# B&R Automation Studio project PT_KB_V01 (part 4)

#### FBAI01_DI01_DO2.st
```iecst
FUNCTION_BLOCK FBAI01_DI01_DO02 (* Skaliranje transmitera sa AI + status DI + 2 DO izbora opsega *) (*$GROUP=User,$CAT=User,$GROUPICON=User.png,$CATICON=User.png*)

(* -------------------------------------------------------------------------- *)
(* 1) Podrazumevane vrednosti po scan-u                                        *)
(* -------------------------------------------------------------------------- *)
(* Podrazumevane vrednosti po scan-u. *)
AI_Output.Status := FALSE;
AI_Internal.FaultCondition := FALSE;
AI_Internal.FaultProcess := FALSE;
AI_Internal.FaultConfig := FALSE;
AI_Output.UnitOfMeasureOut := AI_Param.UnitOfMeasure;
AI_Output.TransmitterStatusIn := AI_Input.TransmitterStatus;
AI_Output.RangeChanging := FALSE;
AI_Output.FaultProcessOut := FALSE;
AI_Output.FaultConfigOut := FALSE;
AI_Internal.ResetRequest := AI_Input.ResetAlarm;

(* -------------------------------------------------------------------------- *)
(* 2) Reset i detekcija promene opsega                                         *)
(* -------------------------------------------------------------------------- *)
(* Eksplicitni reset latched alarma. *)
IF AI_Internal.ResetRequest THEN
	AI_Internal.FaultLatched := FALSE;
END_IF;

(* Detekcija promene opsega. *)
IF AI_Input.RangeSelect <> AI_Internal.PrevRangeSelect THEN
	AI_Internal.RangeChangeMem := TRUE;
END_IF;

(* -------------------------------------------------------------------------- *)
(* 3) Izbor opsega i mapiranje DO bitova                                       *)
(* -------------------------------------------------------------------------- *)
(* Izbor aktivnog opsega i mapiranje u 2 izlazna DO bita. *)
CASE AI_Input.RangeSelect OF
	1:
		AI_Output.ActiveRange := 1;
		AI_Output.RangeBit0_out := FALSE;
		AI_Output.RangeBit1_out := FALSE;
		AI_Internal.ActiveScaledMin := AI_Param.ScaledMin_R1;
		AI_Internal.ActiveScaledMax := AI_Param.ScaledMax_R1;
		AI_Output.RangeComment := 'Opseg 1';
	2:
		AI_Output.ActiveRange := 2;
		AI_Output.RangeBit0_out := TRUE;
		AI_Output.RangeBit1_out := FALSE;
		AI_Internal.ActiveScaledMin := AI_Param.ScaledMin_R2;
		AI_Internal.ActiveScaledMax := AI_Param.ScaledMax_R2;
		AI_Output.RangeComment := 'Opseg 2';
	3:
		AI_Output.ActiveRange := 3;
		AI_Output.RangeBit0_out := FALSE;
		AI_Output.RangeBit1_out := TRUE;
		AI_Internal.ActiveScaledMin := AI_Param.ScaledMin_R3;
		AI_Internal.ActiveScaledMax := AI_Param.ScaledMax_R3;
		AI_Output.RangeComment := 'Opseg 3';
	4:
		AI_Output.ActiveRange := 4;
		AI_Output.RangeBit0_out := TRUE;
		AI_Output.RangeBit1_out := TRUE;
		AI_Internal.ActiveScaledMin := AI_Param.ScaledMin_R4;
		AI_Internal.ActiveScaledMax := AI_Param.ScaledMax_R4;
		AI_Output.RangeComment := 'Opseg 4';
	ELSE
		AI_Output.ActiveRange := 1;
		AI_Output.RangeBit0_out := FALSE;
		AI_Output.RangeBit1_out := FALSE;
		AI_Internal.ActiveScaledMin := AI_Param.ScaledMin_R1;
		AI_Internal.ActiveScaledMax := AI_Param.ScaledMax_R1;
		AI_Output.RangeComment := 'Nevalidan opseg';
		AI_Internal.FaultConfig := TRUE;
END_CASE;

(* -------------------------------------------------------------------------- *)
(* 4) Ogranicenje manual vrednosti i range-settle tajmer                       *)
(* -------------------------------------------------------------------------- *)
(* Ogranicenje manual vrednosti na aktivni opseg. *)
AI_Internal.ManualValueLimited := AI_Input.ManualValue;
IF AI_Internal.ManualValueLimited < AI_Internal.ActiveScaledMin THEN
	AI_Internal.ManualValueLimited := AI_Internal.ActiveScaledMin;
END_IF;
IF AI_Internal.ManualValueLimited > AI_Internal.ActiveScaledMax THEN
	AI_Internal.ManualValueLimited := AI_Internal.ActiveScaledMax;
END_IF;

(* Tajmer stabilizacije nakon promene opsega. *)
AI_Internal.RangeSettleTimeEffective := AI_Input.RangeSettleTime;
IF AI_Internal.RangeSettleTimeEffective <= T#0ms THEN
	AI_Internal.RangeSettleTimeEffective := T#2s;
	AI_Internal.FaultConfig := TRUE;
END_IF;

AI_Internal.RangeSettleTimer(
	IN := AI_Internal.RangeChangeMem,
	PT := AI_Internal.RangeSettleTimeEffective
);
AI_Output.RangeChanging := AI_Internal.RangeChangeMem;
IF AI_Internal.RangeSettleTimer.Q THEN
	AI_Internal.RangeChangeMem := FALSE;
END_IF;

(* -------------------------------------------------------------------------- *)
(* 5) Glavna obrada kada je blok omogucen                                      *)
(* -------------------------------------------------------------------------- *)
IF NOT AI_Input.Enable THEN
	AI_Output.ScaledValue := 0.0;
	AI_Output.State := AI_Constant.ST_DISABLED;
	AI_Output.State_comment := AI_Constant.CMT_DISABLED;
	AI_Output.Status := FALSE;
ELSE
	(* Racunanje raspona za linearnu transformaciju raw -> scaled. *)
	AI_Internal.ScaleSpanRaw := INT_TO_REAL(AI_Param.RawMax - AI_Param.RawMin);
	AI_Internal.ScaleSpanScaled := AI_Internal.ActiveScaledMax - AI_Internal.ActiveScaledMin;

	IF AI_Internal.ScaleSpanRaw <= 0.0 THEN
		AI_Internal.FaultConfig := TRUE;
	END_IF;

	IF AI_Internal.ScaleSpanScaled <= 0.0 THEN
		AI_Internal.FaultConfig := TRUE;
	END_IF;

	IF AI_Input.ManualAlarm THEN
		AI_Internal.FaultProcess := TRUE;
	END_IF;

	IF NOT AI_Output.RangeChanging THEN
		IF AI_Input.UnderRange OR AI_Input.OverRange THEN
			AI_Internal.FaultProcess := TRUE;
		END_IF;

		IF NOT AI_Input.TransmitterStatus THEN
			AI_Internal.FaultProcess := TRUE;
		END_IF;
	END_IF;

	IF AI_Output.RangeChanging THEN
		AI_Output.ScaledValue := AI_Internal.LastGoodScaledValue;
	ELSIF AI_Input.EnableManual THEN
		AI_Output.ScaledValue := AI_Internal.ManualValueLimited;
		AI_Internal.LastGoodScaledValue := AI_Output.ScaledValue;
	ELSE
		IF AI_Internal.ScaleSpanRaw > 0.0 THEN
			AI_Output.ScaledValue :=
				AI_Internal.ActiveScaledMin +
				((INT_TO_REAL(AI_Input.RawValue - AI_Param.RawMin) / AI_Internal.ScaleSpanRaw) * AI_Internal.ScaleSpanScaled);
			AI_Internal.LastGoodScaledValue := AI_Output.ScaledValue;
		ELSE
			AI_Output.ScaledValue := AI_Internal.ActiveScaledMin;
		END_IF;
	END_IF;

	AI_Internal.FaultCondition := AI_Internal.FaultProcess OR AI_Internal.FaultConfig;
	AI_Output.FaultProcessOut := AI_Internal.FaultProcess;
	AI_Output.FaultConfigOut := AI_Internal.FaultConfig;

	IF AI_Internal.FaultCondition THEN
		AI_Internal.FaultLatched := TRUE;
	END_IF;

	(* ---------------------------------------------------------------------- *)
	(* 6) State i status mapiranje                                             *)
	(* ---------------------------------------------------------------------- *)
	IF AI_Output.RangeChanging THEN
		AI_Output.State := AI_Constant.ST_RANGE_CHANGING;
		AI_Output.State_comment := AI_Constant.CMT_RANGE_CHANGING;
		AI_Output.Status := FALSE;
	ELSIF AI_Internal.FaultLatched AND AI_Input.EnableManual THEN
		AI_Output.State := AI_Constant.ST_MANUAL_FAULT;
		AI_Output.State_comment := AI_Constant.CMT_MANUAL_FAULT;
		AI_Output.Status := FALSE;
	ELSIF AI_Input.EnableManual THEN
		AI_Output.State := AI_Constant.ST_MANUAL;
		AI_Output.State_comment := AI_Constant.CMT_MANUAL;
		AI_Output.Status := AI_Input.TransmitterStatus;
	ELSIF AI_Internal.FaultLatched THEN
		AI_Output.State := AI_Constant.ST_FAULT;
		AI_Output.State_comment := AI_Constant.CMT_FAULT;
		AI_Output.Status := FALSE;
	ELSIF NOT AI_Input.TransmitterStatus THEN
		AI_Output.State := AI_Constant.ST_TRANSMITTER_STATUS_0;
		AI_Output.State_comment := AI_Constant.CMT_TRANSMITTER_STATUS_0;
		AI_Output.Status := FALSE;
	ELSIF AI_Input.RawValue < AI_Param.RawMin THEN
		AI_Output.State := AI_Constant.ST_UNDERRANGE;
		AI_Output.State_comment := AI_Constant.CMT_UNDERRANGE;
		AI_Output.Status := FALSE;
	ELSIF AI_Input.RawValue > AI_Param.RawMax THEN
		AI_Output.State := AI_Constant.ST_OVERRANGE;
		AI_Output.State_comment := AI_Constant.CMT_OVERRANGE;
		AI_Output.Status := FALSE;
	ELSE
		AI_Output.State := AI_Constant.ST_ACTIVE;
		AI_Output.State_comment := AI_Constant.CMT_ACTIVE;
		AI_Output.Status := TRUE;
	END_IF;
END_IF;

(* -------------------------------------------------------------------------- *)
(* 7) Pamcenje prethodnog opsega za sledeci scan                               *)
(* -------------------------------------------------------------------------- *)
(* Pamcenje prethodnog opsega. *)
AI_Internal.PrevRangeSelect := AI_Input.RangeSelect;

END_FUNCTION_BLOCK
```

#### FB_PvAiAo_Fast.st
```iecst
FUNCTION_BLOCK FB_PvAiAo_Fast

(* Preporuka za commissioning (nije automatsko prepisivanje parametara):
	DeviationOnLimit = 8.0
	DeviationOffLimit = 3.0
	DeviationTime = T#5s
*)

(* -------------------------------------------------------------------------- *)
(* 1) Osnovni statusi bloka                                                    *)
(* -------------------------------------------------------------------------- *)
PV_Output.Valid := PV_Input.Enable;
PV_Output.ManualActive := PV_Input.EnableManual;

(* -------------------------------------------------------------------------- *)
(* 2) Ogranicenje AI ulaza i skaliranje u procente                             *)
(* -------------------------------------------------------------------------- *)
IF PV_Input.AI_Raw < PV_Constant.RAW_MIN THEN
	PV_Output.AI_Raw_Limited := PV_Constant.RAW_MIN;
ELSIF PV_Input.AI_Raw > PV_Constant.RAW_MAX THEN
	PV_Output.AI_Raw_Limited := PV_Constant.RAW_MAX;
ELSE
	PV_Output.AI_Raw_Limited := PV_Input.AI_Raw;
END_IF;

PV_Internal.rAi := INT_TO_REAL(PV_Output.AI_Raw_Limited);
PV_Output.PV_Percent := (PV_Internal.rAi * PV_Constant.PCT_MAX) / INT_TO_REAL(PV_Constant.RAW_MAX);

(* -------------------------------------------------------------------------- *)
(* 3) Ogranicenje auto i manual komande                                        *)
(* -------------------------------------------------------------------------- *)
IF PV_Input.SP_Percent < PV_Constant.PCT_MIN THEN
	PV_Output.SP_Percent_Limited := PV_Constant.PCT_MIN;
ELSIF PV_Input.SP_Percent > PV_Constant.PCT_MAX THEN
	PV_Output.SP_Percent_Limited := PV_Constant.PCT_MAX;
ELSE
	PV_Output.SP_Percent_Limited := PV_Input.SP_Percent;
END_IF;

IF PV_Input.ManualValue_Percent < PV_Constant.PCT_MIN THEN
	PV_Output.ManualValue_Limited := PV_Constant.PCT_MIN;
ELSIF PV_Input.ManualValue_Percent > PV_Constant.PCT_MAX THEN
	PV_Output.ManualValue_Limited := PV_Constant.PCT_MAX;
ELSE
	PV_Output.ManualValue_Limited := PV_Input.ManualValue_Percent;
END_IF;

(* -------------------------------------------------------------------------- *)
(* 4) Izbor aktivne komande (manual ima prioritet)                             *)
(* -------------------------------------------------------------------------- *)
IF PV_Input.EnableManual THEN
	PV_Output.ActiveSP_Limited := PV_Output.ManualValue_Limited;
ELSE
	PV_Output.ActiveSP_Limited := PV_Output.SP_Percent_Limited;
END_IF;
PV_Output.ActiveSP_Percent := PV_Output.ActiveSP_Limited;

(* -------------------------------------------------------------------------- *)
(* 5) Validacija devijacionih granica i vremena                                *)
(* -------------------------------------------------------------------------- *)
IF PV_Param.DeviationOnLimit < PV_Constant.PCT_MIN THEN
	PV_Output.DeviationOn_Limited := PV_Constant.PCT_MIN;
ELSIF PV_Param.DeviationOnLimit > PV_Constant.PCT_MAX THEN
	PV_Output.DeviationOn_Limited := PV_Constant.PCT_MAX;
ELSE
	PV_Output.DeviationOn_Limited := PV_Param.DeviationOnLimit;
END_IF;

IF PV_Param.DeviationOffLimit < PV_Constant.PCT_MIN THEN
	PV_Output.DeviationOff_Limited := PV_Constant.PCT_MIN;
ELSIF PV_Param.DeviationOffLimit > PV_Constant.PCT_MAX THEN
	PV_Output.DeviationOff_Limited := PV_Constant.PCT_MAX;
ELSE
	PV_Output.DeviationOff_Limited := PV_Param.DeviationOffLimit;
END_IF;

IF PV_Output.DeviationOff_Limited > PV_Output.DeviationOn_Limited THEN
	PV_Output.DeviationOff_Limited := PV_Output.DeviationOn_Limited;
END_IF;

IF PV_Param.DeviationTime <= T#0ms THEN
	PV_Output.DeviationTime_Effective := PV_Constant.MIN_DEV_TIME;
ELSE
	PV_Output.DeviationTime_Effective := PV_Param.DeviationTime;
END_IF;

(* -------------------------------------------------------------------------- *)
(* 6) Proracun devijacije i tolerancije                                        *)
(* -------------------------------------------------------------------------- *)
PV_Output.DeviationPercent := ABS(PV_Output.ActiveSP_Limited - PV_Output.PV_Percent);
PV_Output.InTolerance := (PV_Output.DeviationPercent <= PV_Output.DeviationOff_Limited);

(* -------------------------------------------------------------------------- *)
(* 7) Fault/reset/deviation stanje i tajmer                                     *)
(* -------------------------------------------------------------------------- *)
IF PV_Input.Reset THEN
	PV_Output.FaultActive := FALSE;
	PV_Output.DeviationTimeout := FALSE;
	PV_Output.InDeviation := FALSE;

	PV_Internal.FB_DeviationTimer.PT := PV_Output.DeviationTime_Effective;
	PV_Internal.FB_DeviationTimer.IN := FALSE;
	PV_Internal.FB_DeviationTimer();
	PV_Output.DeviationElapsed := PV_Internal.FB_DeviationTimer.ET;

ELSIF NOT PV_Input.Enable THEN
	PV_Output.InDeviation := FALSE;

	PV_Internal.FB_DeviationTimer.PT := PV_Output.DeviationTime_Effective;
	PV_Internal.FB_DeviationTimer.IN := FALSE;
	PV_Internal.FB_DeviationTimer();
	PV_Output.DeviationElapsed := PV_Internal.FB_DeviationTimer.ET;

ELSE
	IF PV_Output.FaultActive THEN
		PV_Output.InDeviation := FALSE;

		PV_Internal.FB_DeviationTimer.PT := PV_Output.DeviationTime_Effective;
		PV_Internal.FB_DeviationTimer.IN := FALSE;
		PV_Internal.FB_DeviationTimer();
		PV_Output.DeviationElapsed := PV_Internal.FB_DeviationTimer.ET;
	ELSE
		IF NOT PV_Output.InDeviation THEN
			IF PV_Output.DeviationPercent >= PV_Output.DeviationOn_Limited THEN
				PV_Output.InDeviation := TRUE;
			END_IF;
		ELSE
			IF PV_Output.DeviationPercent <= PV_Output.DeviationOff_Limited THEN
				PV_Output.InDeviation := FALSE;
			END_IF;
		END_IF;

		PV_Internal.FB_DeviationTimer.PT := PV_Output.DeviationTime_Effective;
		PV_Internal.FB_DeviationTimer.IN := PV_Output.InDeviation;
		PV_Internal.FB_DeviationTimer();
		PV_Output.DeviationElapsed := PV_Internal.FB_DeviationTimer.ET;

		IF PV_Output.InDeviation AND PV_Internal.FB_DeviationTimer.Q THEN
			PV_Output.FaultActive := TRUE;
			PV_Output.DeviationTimeout := TRUE;
			PV_Output.InDeviation := FALSE;
		END_IF;
	END_IF;
END_IF;

(* -------------------------------------------------------------------------- *)
(* 8) Izbor stvarno primenjene izlazne komande                                  *)
(* -------------------------------------------------------------------------- *)
IF NOT PV_Input.Enable THEN
	PV_Output.AppliedOutput_Limited := PV_Constant.PCT_MIN;
	PV_Output.FrozenOutput_Percent := PV_Constant.PCT_MIN;
	PV_Output.CommandPermitted := FALSE;
	PV_Output.ForceActive := FALSE;

ELSIF PV_Output.FaultActive THEN
	IF PV_Input.ForceCmd THEN
		PV_Output.AppliedOutput_Limited := PV_Output.ActiveSP_Limited;
		PV_Output.CommandPermitted := TRUE;
		PV_Output.ForceActive := TRUE;
	ELSE
		PV_Output.CommandPermitted := FALSE;
		PV_Output.ForceActive := FALSE;

		IF PV_Param.HoldOutputOnFault THEN
			PV_Output.AppliedOutput_Limited := PV_Output.FrozenOutput_Percent;
		ELSE
			PV_Output.AppliedOutput_Limited := PV_Constant.PCT_MIN;
		END_IF;
	END_IF;
ELSE
	PV_Output.AppliedOutput_Limited := PV_Output.ActiveSP_Limited;
	PV_Output.CommandPermitted := TRUE;
	PV_Output.ForceActive := FALSE;
	PV_Output.FrozenOutput_Percent := PV_Output.AppliedOutput_Limited;
END_IF;

(* -------------------------------------------------------------------------- *)
(* 9) Zavrsno ogranicenje i AO skaliranje                                      *)
(* -------------------------------------------------------------------------- *)
IF PV_Output.AppliedOutput_Limited < PV_Constant.PCT_MIN THEN
	PV_Output.AppliedOutput_Limited := PV_Constant.PCT_MIN;
ELSIF PV_Output.AppliedOutput_Limited > PV_Constant.PCT_MAX THEN
	PV_Output.AppliedOutput_Limited := PV_Constant.PCT_MAX;
END_IF;
PV_Output.AppliedOutput_Percent := PV_Output.AppliedOutput_Limited;

PV_Internal.rAo := (PV_Output.AppliedOutput_Limited * INT_TO_REAL(PV_Constant.RAW_MAX)) / PV_Constant.PCT_MAX;
PV_Internal.AO_Raw_Calc := REAL_TO_INT(PV_Internal.rAo);

IF PV_Internal.AO_Raw_Calc < PV_Constant.RAW_MIN THEN
	PV_Internal.AO_Raw_Calc := PV_Constant.RAW_MIN;
ELSIF PV_Internal.AO_Raw_Calc > PV_Constant.RAW_MAX THEN
	PV_Internal.AO_Raw_Calc := PV_Constant.RAW_MAX;
END_IF;
PV_Output.AO_Raw := PV_Internal.AO_Raw_Calc;

(* -------------------------------------------------------------------------- *)
(* 10) Standardni izlazi stanja za HMI/SCADA                                    *)
(* -------------------------------------------------------------------------- *)
IF NOT PV_Input.Enable THEN
	PV_Output.Status := FALSE;
	PV_Output.State := PV_Constant.ST_DISABLED;
	PV_Output.State_comment := 'ST_DISABLED - blok nije omogucen';
ELSIF PV_Output.FaultActive THEN
	PV_Output.Status := FALSE;
	IF PV_Output.ForceActive THEN
		PV_Output.State := PV_Constant.ST_FAULT_FORCE;
		PV_Output.State_comment := 'ST_FAULT_FORCE - fault aktivan, izlaz forsiran';
	ELSE
		PV_Output.State := PV_Constant.ST_FAULT_HOLD;
		PV_Output.State_comment := 'ST_FAULT_HOLD - fault aktivan, izlaz blokiran/hold';
	END_IF;
ELSIF PV_Output.InDeviation THEN
	PV_Output.Status := TRUE;
	PV_Output.State := PV_Constant.ST_DEVIATION_ACTIVE;
	PV_Output.State_comment := 'ST_DEVIATION_ACTIVE - aktivno pracenje devijacije';
ELSIF PV_Output.ManualActive THEN
	PV_Output.Status := TRUE;
	PV_Output.State := PV_Constant.ST_MANUAL_ACTIVE;
	PV_Output.State_comment := 'ST_MANUAL_ACTIVE - aktivan manuelni rezim';
ELSE
	PV_Output.Status := TRUE;
	PV_Output.State := PV_Constant.ST_AUTO_ACTIVE;
	PV_Output.State_comment := 'ST_AUTO_ACTIVE - aktivan automatski rezim';
END_IF;

END_FUNCTION_BLOCK
```

#### FB_PvAiAo_Slow.st
```iecst
(* SLOW VARIJANTA: Za elektromotorne ventile sa sporim odzivom (30-180 s). *)
(* Implementirana logika: trenutna komanda + nadzor fizickog pracenja ventila. *)

(*
===============================================================================
SLOW LOGIC SPEC (USAGLASENO PRE IMPLEMENTACIJE)
===============================================================================

Osnovni princip:
1) Komanda izlaza se NE rampira softverski.
2) Kada se promeni setpoint, izlaz odmah dobija novu komandnu vrednost.
3) Umesto rampe proverava se da li ventil fizicki prati ocekivano vreme putovanja.

Definicije:
- PV_Internal.StepDeltaPercent = ABS(NewSP - PV_Internal.PrevSP)
- Smer kretanja:
	- Opening: NewSP > PV_Internal.PrevSP
	- Closing: NewSP < PV_Internal.PrevSP
- Ocekivano vreme putovanja:
	- Texp_open  = PV_Internal.StepDeltaPercent/100 * PV_Internal.TravelTimeOpenFull
	- Texp_close = PV_Internal.StepDeltaPercent/100 * PV_Internal.TravelTimeCloseFull
- Dozvoljeni prozor:
	- Tmin = Texp * (1 - PV_Internal.TimeTolerancePercent/100)
	- Tmax = Texp * (1 + PV_Internal.TimeTolerancePercent/100)

Ulaz u tracking poteza:
- Tracking se aktivira kada je ABS(NewSP - PV_Internal.PrevSP) >= StepMinPercent.
- Ako je manji korak od StepMinPercent, tretira se kao mali pomak bez punog timing nadzora.

Uslovi tokom tracking-a:
1) Start movement timeout:
	 - Ako nema detektovanog pocetnog pomeranja PV u PV_Internal.StartMoveTimeout -> FaultNoMovement.
2) Smer kretanja:
	 - Opening: PV mora da raste.
	 - Closing: PV mora da opada.
	 - Suprotan smer duze od PV_Internal.DirectionCheckTime -> FaultWrongDirection.
3) Stall nadzor:
	 - Ako je tracking aktivan, a PV ne menja vrednost duze od PV_Internal.StallTimeout -> FaultStall.
4) Zavrsetak poteza:
	 - Potez je zavrsen kada PV udje u ciljnu traku:
		 ABS(TargetSP - PV) <= TargetBandPercent.
	 - Ako zavrsetak nastupi pre Tmin -> warning ili fault (po parametru PV_Internal.EnableTooFastFault).
	 - Ako zavrsetak ne nastupi do Tmax -> FaultTimeout.

Nova komanda tokom aktivnog poteza:
- Aktivni tracking se prekida i odmah se formira novi tracking od trenutnog PV/SP stanja.

Fault politika:
- Fault je latched (ostaje aktivan do Reset).
- Fault tipovi:
	1) NoMovement
	2) WrongDirection
	3) Stall
	4) TimeoutSlow
	5) (opciono) TooFast

Interakcija sa postojecim logikama:
- Enable i dalje ima apsolutni prioritet (disable gasi komandu).
- ForceCmd i HoldOutputOnFault zadrzavaju isto ponasanje kao FAST varijanta.
- Status/State/State_comment ostaju obavezni izlazi.

Napomena za implementaciju:
- Uvesti odvojene interne tajmere za:
	- start movement timeout,
	- direction confirm,
	- stall timeout,
	- tracking timeout (Tmax).
- Uvesti internu memoriju prethodnog SP i prethodnog PV za detekciju koraka i trenda.
===============================================================================
*)

FUNCTION_BLOCK FB_PvAiAo_Slow

(* Commissioning preset (pocetne preporuke, po potrebi menjati na terenu):
   PV_Internal.TravelTimeOpenFull = T#120s
   PV_Internal.TravelTimeCloseFull = T#120s
   PV_Internal.TimeTolerancePercent = 35.0
   PV_Internal.StartMoveTimeout = T#8s
   PV_Internal.DirectionCheckTime = T#8s
   PV_Internal.StallTimeout = T#20s
   PV_Internal.MovementStartDeltaPercent = 0.7
   PV_Internal.PerScanProgressMinPercent = 0.03
   PV_Internal.DirectionEpsPercent = 0.03
   PV_Internal.EnableTooFastFault = FALSE
*)

(* -------------------------------------------------------------------------- *)
(* 1) Osnovni statusi bloka                                                    *)
(* -------------------------------------------------------------------------- *)
PV_Output.Valid := PV_Input.Enable;
PV_Output.ManualActive := PV_Input.EnableManual;

(* -------------------------------------------------------------------------- *)
(* 2) Ogranicenje AI ulaza i skaliranje u procente                             *)
(* -------------------------------------------------------------------------- *)
IF PV_Input.AI_Raw < PV_Constant.RAW_MIN THEN
	PV_Output.AI_Raw_Limited := PV_Constant.RAW_MIN;
ELSIF PV_Input.AI_Raw > PV_Constant.RAW_MAX THEN
	PV_Output.AI_Raw_Limited := PV_Constant.RAW_MAX;
ELSE
	PV_Output.AI_Raw_Limited := PV_Input.AI_Raw;
END_IF;

PV_Internal.rAi := INT_TO_REAL(PV_Output.AI_Raw_Limited);
PV_Output.PV_Percent := (PV_Internal.rAi * PV_Constant.PCT_MAX) / INT_TO_REAL(PV_Constant.RAW_MAX);

(* -------------------------------------------------------------------------- *)
(* 3) Ogranicenje auto i manual komande                                        *)
(* -------------------------------------------------------------------------- *)
IF PV_Input.SP_Percent < PV_Constant.PCT_MIN THEN
	PV_Output.SP_Percent_Limited := PV_Constant.PCT_MIN;
ELSIF PV_Input.SP_Percent > PV_Constant.PCT_MAX THEN
	PV_Output.SP_Percent_Limited := PV_Constant.PCT_MAX;
ELSE
	PV_Output.SP_Percent_Limited := PV_Input.SP_Percent;
END_IF;

IF PV_Input.ManualValue_Percent < PV_Constant.PCT_MIN THEN
	PV_Output.ManualValue_Limited := PV_Constant.PCT_MIN;
ELSIF PV_Input.ManualValue_Percent > PV_Constant.PCT_MAX THEN
	PV_Output.ManualValue_Limited := PV_Constant.PCT_MAX;
ELSE
	PV_Output.ManualValue_Limited := PV_Input.ManualValue_Percent;
END_IF;

(* -------------------------------------------------------------------------- *)
(* 4) Izbor aktivne komande (manual ima prioritet)                             *)
(* -------------------------------------------------------------------------- *)
IF PV_Input.EnableManual THEN
	PV_Output.ActiveSP_Limited := PV_Output.ManualValue_Limited;
ELSE
	PV_Output.ActiveSP_Limited := PV_Output.SP_Percent_Limited;
END_IF;
PV_Output.ActiveSP_Percent := PV_Output.ActiveSP_Limited;

(* -------------------------------------------------------------------------- *)
(* 5) Validacija devijacionih granica i vremena                                *)
(* -------------------------------------------------------------------------- *)
IF PV_Param.DeviationOnLimit < PV_Constant.PCT_MIN THEN
	PV_Output.DeviationOn_Limited := PV_Constant.PCT_MIN;
ELSIF PV_Param.DeviationOnLimit > PV_Constant.PCT_MAX THEN
	PV_Output.DeviationOn_Limited := PV_Constant.PCT_MAX;
ELSE
	PV_Output.DeviationOn_Limited := PV_Param.DeviationOnLimit;
END_IF;

IF PV_Param.DeviationOffLimit < PV_Constant.PCT_MIN THEN
	PV_Output.DeviationOff_Limited := PV_Constant.PCT_MIN;
ELSIF PV_Param.DeviationOffLimit > PV_Constant.PCT_MAX THEN
	PV_Output.DeviationOff_Limited := PV_Constant.PCT_MAX;
ELSE
	PV_Output.DeviationOff_Limited := PV_Param.DeviationOffLimit;
END_IF;

IF PV_Output.DeviationOff_Limited > PV_Output.DeviationOn_Limited THEN
	PV_Output.DeviationOff_Limited := PV_Output.DeviationOn_Limited;
END_IF;

IF PV_Param.DeviationTime <= T#0ms THEN
	PV_Output.DeviationTime_Effective := PV_Constant.MIN_DEV_TIME;
ELSE
	PV_Output.DeviationTime_Effective := PV_Param.DeviationTime;
END_IF;

(* -------------------------------------------------------------------------- *)
(* 6) Proracun devijacije i tolerancije                                        *)
(* -------------------------------------------------------------------------- *)
PV_Output.DeviationPercent := ABS(PV_Output.ActiveSP_Limited - PV_Output.PV_Percent);
PV_Output.InTolerance := (PV_Output.DeviationPercent <= PV_Output.DeviationOff_Limited);

(* -------------------------------------------------------------------------- *)
(* 7) Tracking i fault nadzor za SLOW ponasanje                                *)
(* -------------------------------------------------------------------------- *)
(* Reset/safe defaults za tracking i fault nadzor. *)
IF PV_Input.Reset THEN
	PV_Output.FaultActive := FALSE;
	PV_Output.DeviationTimeout := FALSE;
	PV_Internal.TrackActive := FALSE;
	PV_Internal.MovementStarted := FALSE;
	PV_Internal.FaultReasonText := 'RESET';
	PV_Output.InDeviation := FALSE;

	PV_Internal.TrackTimer(IN := FALSE, PT := T#1ms);
	PV_Internal.StartMoveTimer(IN := FALSE, PT := PV_Internal.StartMoveTimeout);
	PV_Internal.DirectionTimer(IN := FALSE, PT := PV_Internal.DirectionCheckTime);
	PV_Internal.StallTimer(IN := FALSE, PT := PV_Internal.StallTimeout);

ELSIF NOT PV_Input.Enable THEN
	PV_Internal.TrackActive := FALSE;
	PV_Internal.MovementStarted := FALSE;
	PV_Output.InDeviation := FALSE;
	PV_Internal.FaultReasonText := 'DISABLED';

	PV_Internal.TrackTimer(IN := FALSE, PT := T#1ms);
	PV_Internal.StartMoveTimer(IN := FALSE, PT := PV_Internal.StartMoveTimeout);
	PV_Internal.DirectionTimer(IN := FALSE, PT := PV_Internal.DirectionCheckTime);
	PV_Internal.StallTimer(IN := FALSE, PT := PV_Internal.StallTimeout);

ELSE
	(* Novo pracenje na znacajnu promenu komande.
	   Prag za aktivaciju tracking-a je vezan za DeviationOn_Limited. *)
	PV_Internal.StepDeltaPercent := ABS(PV_Output.ActiveSP_Limited - PV_Internal.PrevSP);
	IF PV_Internal.StepDeltaPercent >= PV_Output.DeviationOn_Limited THEN
		PV_Internal.TrackActive := TRUE;
		PV_Internal.MovementStarted := FALSE;
		PV_Internal.PV_AtTrackStart := PV_Output.PV_Percent;
		PV_Internal.LastProgressPV := PV_Output.PV_Percent;
		PV_Internal.TrackDirectionOpen := (PV_Output.ActiveSP_Limited > PV_Internal.PrevSP);

		IF PV_Internal.TrackDirectionOpen THEN
			PV_Internal.ExpectedTravelSec := (PV_Internal.StepDeltaPercent / 100.0) * (TIME_TO_REAL(PV_Internal.TravelTimeOpenFull) / 1000.0);
		ELSE
			PV_Internal.ExpectedTravelSec := (PV_Internal.StepDeltaPercent / 100.0) * (TIME_TO_REAL(PV_Internal.TravelTimeCloseFull) / 1000.0);
		END_IF;

		PV_Internal.TminSec := PV_Internal.ExpectedTravelSec * (1.0 - PV_Internal.TimeTolerancePercent / 100.0);
		PV_Internal.TmaxSec := PV_Internal.ExpectedTravelSec * (1.0 + PV_Internal.TimeTolerancePercent / 100.0);
		IF PV_Internal.TminSec < 0.0 THEN
			PV_Internal.TminSec := 0.0;
		END_IF;
		IF PV_Internal.TmaxSec <= 0.0 THEN
			PV_Internal.TmaxSec := 0.1;
		END_IF;
	END_IF;

	(* Tajmeri nadzora putovanja. *)
	PV_Internal.TrackTimer(IN := PV_Internal.TrackActive, PT := REAL_TO_TIME(PV_Internal.TmaxSec * 1000.0));
	PV_Internal.StartMoveTimer(IN := PV_Internal.TrackActive AND (NOT PV_Internal.MovementStarted), PT := PV_Internal.StartMoveTimeout);

	IF PV_Internal.TrackActive THEN
		IF ABS(PV_Output.PV_Percent - PV_Internal.PV_AtTrackStart) >= PV_Internal.MovementStartDeltaPercent THEN
			PV_Internal.MovementStarted := TRUE;
		END_IF;

		IF PV_Internal.TrackDirectionOpen THEN
			PV_Internal.DirectionTimer(IN := (PV_Output.PV_Percent < (PV_Internal.PrevPV - PV_Internal.DirectionEpsPercent)), PT := PV_Internal.DirectionCheckTime);
		ELSE
			PV_Internal.DirectionTimer(IN := (PV_Output.PV_Percent > (PV_Internal.PrevPV + PV_Internal.DirectionEpsPercent)), PT := PV_Internal.DirectionCheckTime);
		END_IF;

		PV_Internal.StallTimer(IN := PV_Internal.MovementStarted AND (ABS(PV_Output.PV_Percent - PV_Internal.PrevPV) < PV_Internal.PerScanProgressMinPercent), PT := PV_Internal.StallTimeout);
	ELSE
		PV_Internal.DirectionTimer(IN := FALSE, PT := PV_Internal.DirectionCheckTime);
		PV_Internal.StallTimer(IN := FALSE, PT := PV_Internal.StallTimeout);
	END_IF;

	(* Fault uslovi i zavrsetak tracking-a. *)
	PV_Output.DeviationTimeout := FALSE;
	IF PV_Internal.TrackActive THEN
		IF PV_Internal.StartMoveTimer.Q THEN
			PV_Output.FaultActive := TRUE;
			PV_Internal.FaultReasonText := 'FAULT_NO_MOVEMENT';
			PV_Internal.TrackActive := FALSE;
		ELSIF PV_Internal.DirectionTimer.Q THEN
			PV_Output.FaultActive := TRUE;
			PV_Internal.FaultReasonText := 'FAULT_WRONG_DIRECTION';
			PV_Internal.TrackActive := FALSE;
		ELSIF PV_Internal.StallTimer.Q THEN
			PV_Output.FaultActive := TRUE;
			PV_Internal.FaultReasonText := 'FAULT_STALL';
			PV_Internal.TrackActive := FALSE;
		ELSIF PV_Internal.TrackTimer.Q THEN
			PV_Output.FaultActive := TRUE;
			PV_Output.DeviationTimeout := TRUE;
			PV_Internal.FaultReasonText := 'FAULT_TIMEOUT_SLOW';
			PV_Internal.TrackActive := FALSE;
		ELSIF PV_Output.InTolerance THEN
			PV_Internal.ActualTravelSec := TIME_TO_REAL(PV_Internal.TrackTimer.ET) / 1000.0;
			IF PV_Internal.EnableTooFastFault AND (PV_Internal.ActualTravelSec < PV_Internal.TminSec) THEN
				PV_Output.FaultActive := TRUE;
				PV_Internal.FaultReasonText := 'FAULT_TOO_FAST';
			ELSE
				PV_Internal.FaultReasonText := 'TRACK_OK';
			END_IF;
			PV_Internal.TrackActive := FALSE;
		END_IF;
	END_IF;

	PV_Output.InDeviation := PV_Internal.TrackActive;
END_IF;

PV_Output.DeviationElapsed := PV_Internal.TrackTimer.ET;

(* -------------------------------------------------------------------------- *)
(* 8) Izbor stvarno primenjene izlazne komande                                  *)
(* -------------------------------------------------------------------------- *)
(* Immediate command (bez rampe), sa istom fault politikom kao FAST. *)
IF NOT PV_Input.Enable THEN
	PV_Output.AppliedOutput_Limited := PV_Constant.PCT_MIN;
	PV_Output.FrozenOutput_Percent := PV_Constant.PCT_MIN;
	PV_Output.CommandPermitted := FALSE;
	PV_Output.ForceActive := FALSE;

ELSIF PV_Output.FaultActive THEN
	IF PV_Input.ForceCmd THEN
		PV_Output.AppliedOutput_Limited := PV_Output.ActiveSP_Limited;
		PV_Output.CommandPermitted := TRUE;
		PV_Output.ForceActive := TRUE;
	ELSE
		PV_Output.CommandPermitted := FALSE;
		PV_Output.ForceActive := FALSE;
		IF PV_Param.HoldOutputOnFault THEN
			PV_Output.AppliedOutput_Limited := PV_Output.FrozenOutput_Percent;
		ELSE
			PV_Output.AppliedOutput_Limited := PV_Constant.PCT_MIN;
		END_IF;
	END_IF;

ELSE
	PV_Output.AppliedOutput_Limited := PV_Output.ActiveSP_Limited;
	PV_Output.CommandPermitted := TRUE;
	PV_Output.ForceActive := FALSE;
	PV_Output.FrozenOutput_Percent := PV_Output.AppliedOutput_Limited;
END_IF;

(* -------------------------------------------------------------------------- *)
(* 9) Zavrsno ogranicenje i AO skaliranje                                      *)
(* -------------------------------------------------------------------------- *)
IF PV_Output.AppliedOutput_Limited < PV_Constant.PCT_MIN THEN
	PV_Output.AppliedOutput_Limited := PV_Constant.PCT_MIN;
ELSIF PV_Output.AppliedOutput_Limited > PV_Constant.PCT_MAX THEN
	PV_Output.AppliedOutput_Limited := PV_Constant.PCT_MAX;
END_IF;

PV_Output.AppliedOutput_Percent := PV_Output.AppliedOutput_Limited;
PV_Internal.rAo := (PV_Output.AppliedOutput_Limited * INT_TO_REAL(PV_Constant.RAW_MAX)) / PV_Constant.PCT_MAX;
PV_Internal.AO_Raw_Calc := REAL_TO_INT(PV_Internal.rAo);
IF PV_Internal.AO_Raw_Calc < PV_Constant.RAW_MIN THEN
	PV_Internal.AO_Raw_Calc := PV_Constant.RAW_MIN;
ELSIF PV_Internal.AO_Raw_Calc > PV_Constant.RAW_MAX THEN
	PV_Internal.AO_Raw_Calc := PV_Constant.RAW_MAX;
END_IF;
PV_Output.AO_Raw := PV_Internal.AO_Raw_Calc;

(* -------------------------------------------------------------------------- *)
(* 10) Standardni izlazi stanja za HMI/SCADA                                    *)
(* -------------------------------------------------------------------------- *)
IF NOT PV_Input.Enable THEN
	PV_Output.Status := FALSE;
	PV_Output.State := PV_Constant.ST_DISABLED;
	PV_Output.State_comment := 'ST_DISABLED - blok nije omogucen';
ELSIF PV_Output.FaultActive THEN
	PV_Output.Status := FALSE;
	IF PV_Output.ForceActive THEN
		PV_Output.State := PV_Constant.ST_FAULT_FORCE;
		PV_Output.State_comment := CONCAT('ST_FAULT_FORCE - ', PV_Internal.FaultReasonText);
	ELSE
		PV_Output.State := PV_Constant.ST_FAULT_HOLD;
		PV_Output.State_comment := CONCAT('ST_FAULT_HOLD - ', PV_Internal.FaultReasonText);
	END_IF;
ELSIF PV_Output.InDeviation THEN
	PV_Output.Status := TRUE;
	PV_Output.State := PV_Constant.ST_DEVIATION_ACTIVE;
	PV_Output.State_comment := 'ST_DEVIATION_ACTIVE - tracking travel time';
ELSIF PV_Output.ManualActive THEN
	PV_Output.Status := TRUE;
	PV_Output.State := PV_Constant.ST_MANUAL_ACTIVE;
	PV_Output.State_comment := 'ST_MANUAL_ACTIVE - aktivan manuelni rezim';
ELSE
	PV_Output.Status := TRUE;
	PV_Output.State := PV_Constant.ST_AUTO_ACTIVE;
	PV_Output.State_comment := 'ST_AUTO_ACTIVE - aktivan automatski rezim';
END_IF;

(* -------------------------------------------------------------------------- *)
(* 11) Memorija prethodnog ciklusa za detekciju koraka i trenda                 *)
(* -------------------------------------------------------------------------- *)
PV_Internal.PrevSP := PV_Output.ActiveSP_Limited;
PV_Internal.PrevPV := PV_Output.PV_Percent;

END_FUNCTION_BLOCK
```

#### FB_PvAoNoFb.st
```iecst
FUNCTION_BLOCK FB_PvAoNoFb

(* -------------------------------------------------------------------------- *)
(* 1) Osnovni statusi i izbor rezima                                           *)
(* -------------------------------------------------------------------------- *)
PV_Output.ManualActive := PV_Input.ManualMode;
PV_Output.ForceActive := FALSE;
PV_Output.ParamInvalid := FALSE;

(* -------------------------------------------------------------------------- *)
(* 2) Validacija parametara i priprema efektivnih granica                      *)
(* -------------------------------------------------------------------------- *)
IF (PV_Param.OutMin < PV_Constant.PCT_MIN) OR
   (PV_Param.OutMin > PV_Constant.PCT_MAX) OR
   (PV_Param.OutMax < PV_Constant.PCT_MIN) OR
   (PV_Param.OutMax > PV_Constant.PCT_MAX) OR
   (PV_Param.OutMin >= PV_Param.OutMax) OR
   (PV_Param.RampUp < 0.0) OR
   (PV_Param.RampDown < 0.0) OR
   (PV_Param.OnDelay < T#0ms) OR
   (PV_Param.OffDelay < T#0ms) THEN
	PV_Output.ParamInvalid := TRUE;
END_IF;

IF PV_Output.ParamInvalid THEN
	PV_Output.OutMin_Effective := PV_Constant.PCT_MIN;
	PV_Output.OutMax_Effective := PV_Constant.PCT_MAX;
	PV_Output.RampUp_Effective := PV_Constant.PCT_MAX;
	PV_Output.RampDown_Effective := PV_Constant.PCT_MAX;
	PV_Output.OnDelay_Effective := T#0ms;
	PV_Output.OffDelay_Effective := T#0ms;
ELSE
	PV_Output.OutMin_Effective := PV_Param.OutMin;
	PV_Output.OutMax_Effective := PV_Param.OutMax;

	IF PV_Param.RampUp <= PV_Constant.STEP_MIN THEN
		PV_Output.RampUp_Effective := PV_Constant.PCT_MAX;
	ELSE
		PV_Output.RampUp_Effective := PV_Param.RampUp;
	END_IF;

	IF PV_Param.RampDown <= PV_Constant.STEP_MIN THEN
		PV_Output.RampDown_Effective := PV_Constant.PCT_MAX;
	ELSE
		PV_Output.RampDown_Effective := PV_Param.RampDown;
	END_IF;

	PV_Output.OnDelay_Effective := PV_Param.OnDelay;
	PV_Output.OffDelay_Effective := PV_Param.OffDelay;
END_IF;

(* -------------------------------------------------------------------------- *)
(* 3) Fault latch i reset politika                                              *)
(* -------------------------------------------------------------------------- *)
IF PV_Input.ResetFault AND NOT PV_Output.ParamInvalid THEN
	PV_Output.FaultActive := FALSE;
	PV_Output.FaultCode := PV_Constant.FLT_NONE;
END_IF;

IF PV_Output.ParamInvalid THEN
	PV_Output.FaultActive := TRUE;
	PV_Output.FaultCode := PV_Constant.FLT_PARAM_INVALID;
END_IF;

IF NOT PV_Input.Enable THEN
	PV_Output.ForceActive := FALSE;
END_IF;

(* -------------------------------------------------------------------------- *)
(* 4) Izbor i ogranicenje komandnog cilja                                       *)
(* -------------------------------------------------------------------------- *)
IF PV_Input.ManualMode THEN
	PV_Output.CmdTarget := PV_Input.ManualOut;
ELSE
	PV_Output.CmdTarget := PV_Input.AutoSP;
END_IF;

IF PV_Output.CmdTarget < PV_Constant.PCT_MIN THEN
	PV_Output.CmdTarget := PV_Constant.PCT_MIN;
ELSIF PV_Output.CmdTarget > PV_Constant.PCT_MAX THEN
	PV_Output.CmdTarget := PV_Constant.PCT_MAX;
END_IF;

PV_Output.CmdLimited := PV_Output.CmdTarget;
IF PV_Output.CmdLimited < PV_Output.OutMin_Effective THEN
	PV_Output.CmdLimited := PV_Output.OutMin_Effective;
ELSIF PV_Output.CmdLimited > PV_Output.OutMax_Effective THEN
	PV_Output.CmdLimited := PV_Output.OutMax_Effective;
END_IF;

(* -------------------------------------------------------------------------- *)
(* 5) OnDelay/OffDelay logika bez feedback-a                                   *)
(* -------------------------------------------------------------------------- *)
PV_Internal.RiseRequest := (PV_Output.CmdLimited > (PV_Output.OutMin_Effective + PV_Internal.EpsPercent));
PV_Internal.FallRequest := NOT PV_Internal.RiseRequest;

PV_Internal.OnDelayTimer(IN := (PV_Input.Enable AND PV_Internal.RiseRequest), PT := PV_Output.OnDelay_Effective);
PV_Internal.OffDelayTimer(IN := (PV_Input.Enable AND PV_Internal.FallRequest), PT := PV_Output.OffDelay_Effective);

IF NOT PV_Input.Enable THEN
	PV_Output.CmdDelayed := PV_Constant.PCT_MIN;
ELSIF PV_Internal.RiseRequest THEN
	IF (PV_Output.OnDelay_Effective <= T#0ms) OR PV_Internal.OnDelayTimer.Q THEN
		PV_Output.CmdDelayed := PV_Output.CmdLimited;
	ELSE
		PV_Output.CmdDelayed := PV_Output.OutMin_Effective;
	END_IF;
ELSE
	IF (PV_Output.OffDelay_Effective <= T#0ms) OR PV_Internal.OffDelayTimer.Q THEN
		PV_Output.CmdDelayed := PV_Output.OutMin_Effective;
	ELSE
		PV_Output.CmdDelayed := PV_Internal.CmdWorking;
	END_IF;
END_IF;

(* -------------------------------------------------------------------------- *)
(* 6) Fault reakcija i force/hold ponasanje                                    *)
(* -------------------------------------------------------------------------- *)
IF NOT PV_Input.Enable THEN
	PV_Output.CmdDelayed := PV_Constant.PCT_MIN;
	PV_Output.ForceActive := FALSE;
ELSIF PV_Output.FaultActive THEN
	IF PV_Input.ForceCmd THEN
		PV_Output.ForceActive := TRUE;
	ELSE
		PV_Output.ForceActive := FALSE;
		IF PV_Param.HoldOnFault THEN
			PV_Output.CmdDelayed := PV_Internal.LastHealthyCmd;
		ELSE
			PV_Output.CmdDelayed := PV_Output.OutMin_Effective;
		END_IF;
	END_IF;
END_IF;

(* -------------------------------------------------------------------------- *)
(* 7) Ramp limit komande (po ciklusu)                                          *)
(* -------------------------------------------------------------------------- *)
IF NOT PV_Input.Enable THEN
	PV_Internal.CmdWorking := PV_Constant.PCT_MIN;
ELSE
	IF PV_Output.CmdDelayed > PV_Internal.CmdWorking THEN
		PV_Internal.CmdWorking := PV_Internal.CmdWorking + PV_Output.RampUp_Effective;
		IF PV_Internal.CmdWorking > PV_Output.CmdDelayed THEN
			PV_Internal.CmdWorking := PV_Output.CmdDelayed;
		END_IF;
	ELSIF PV_Output.CmdDelayed < PV_Internal.CmdWorking THEN
		PV_Internal.CmdWorking := PV_Internal.CmdWorking - PV_Output.RampDown_Effective;
		IF PV_Internal.CmdWorking < PV_Output.CmdDelayed THEN
			PV_Internal.CmdWorking := PV_Output.CmdDelayed;
		END_IF;
	END_IF;
END_IF;

IF PV_Internal.CmdWorking < PV_Constant.PCT_MIN THEN
	PV_Internal.CmdWorking := PV_Constant.PCT_MIN;
ELSIF PV_Internal.CmdWorking > PV_Constant.PCT_MAX THEN
	PV_Internal.CmdWorking := PV_Constant.PCT_MAX;
END_IF;

PV_Output.AO_Cmd := PV_Internal.CmdWorking;

IF PV_Input.Enable AND NOT PV_Output.FaultActive THEN
	PV_Internal.LastHealthyCmd := PV_Output.AO_Cmd;
END_IF;

(* -------------------------------------------------------------------------- *)
(* 8) Standardni izlazi stanja                                                 *)
(* -------------------------------------------------------------------------- *)
IF NOT PV_Input.Enable THEN
	PV_Output.Status := FALSE;
	PV_Output.State := PV_Constant.ST_DISABLED;
	PV_Output.State_comment := 'ST_DISABLED - blok nije omogucen';
ELSIF PV_Output.FaultActive THEN
	PV_Output.Status := FALSE;
	IF PV_Output.ForceActive THEN
		PV_Output.State := PV_Constant.ST_FAULT_FORCE;
		PV_Output.State_comment := 'ST_FAULT_FORCE - fault aktivan, izlaz forsiran';
	ELSE
		PV_Output.State := PV_Constant.ST_FAULT_HOLD;
		PV_Output.State_comment := 'ST_FAULT_HOLD - fault aktivan, izlaz hold/zero';
	END_IF;
ELSIF PV_Output.ManualActive THEN
	PV_Output.Status := TRUE;
	PV_Output.State := PV_Constant.ST_MANUAL_ACTIVE;
	PV_Output.State_comment := 'ST_MANUAL_ACTIVE - manuelni rezim';
ELSE
	PV_Output.Status := TRUE;
	PV_Output.State := PV_Constant.ST_AUTO_ACTIVE;
	PV_Output.State_comment := 'ST_AUTO_ACTIVE - automatski rezim';
END_IF;

END_FUNCTION_BLOCK
```

#### FB_AirRelease.st
```iecst
FUNCTION_BLOCK FB_AirRelease (* Automatsko odzracivanje cevovoda sa 1 do 3 LS senzora. *)

(* -------------------------------------------------------------------------- *)
(* 1) Runtime vreme task ciklusa                                               *)
(* -------------------------------------------------------------------------- *)
AR_Internal.RtInfo(enable := TRUE);
AR_Internal.RuntimeTimeValid :=
	(AR_Internal.RtInfo.status = 0)
	AND (AR_Internal.RtInfo.cycle_time > 0)
	AND (AR_Internal.RtInfo.cycle_time <= 1000000);

IF AR_Internal.RuntimeTimeValid THEN
	AR_Output.CycleTime_s := UDINT_TO_REAL(AR_Internal.RtInfo.cycle_time) / 1000000.0;
ELSE
	AR_Output.CycleTime_s := 0.0;
END_IF;

(* -------------------------------------------------------------------------- *)
(* 2) Validacija parametara                                                    *)
(* -------------------------------------------------------------------------- *)
AR_Internal.ConfigValid := TRUE;
AR_Internal.ConfigFaultText := 'CONFIG_OK';

IF (AR_Param.NumberOfLS < 1) OR (AR_Param.NumberOfLS > 3) THEN
	AR_Internal.ConfigValid := FALSE;
	AR_Internal.ConfigFaultText := 'NumberOfLS mora biti u opsegu 1..3';
ELSIF AR_Param.PressureSP_bar < 0.0 THEN
	AR_Internal.ConfigValid := FALSE;
	AR_Internal.ConfigFaultText := 'PressureSP_bar ne sme biti negativan';
ELSIF (AR_Param.PressureHysteresis_bar < 0.0)
	OR (AR_Param.PressureHysteresis_bar > AR_Param.PressureSP_bar) THEN
	AR_Internal.ConfigValid := FALSE;
	AR_Internal.ConfigFaultText := 'PressureHysteresis_bar mora biti 0..PressureSP';
ELSIF (AR_Param.LS1.SP_Percent < AR_Constant.PCT_MIN)
	OR (AR_Param.LS1.SP_Percent > AR_Constant.PCT_MAX) THEN
	AR_Internal.ConfigValid := FALSE;
	AR_Internal.ConfigFaultText := 'LS1 SP mora biti u opsegu 0..100%';
ELSIF AR_Param.LS1.Ramp_PercentPerSecond < AR_Constant.RAMP_MIN THEN
	AR_Internal.ConfigValid := FALSE;
	AR_Internal.ConfigFaultText := 'LS1 rampa mora biti veca od 0%/s';
ELSIF (AR_Param.LS1.ConfirmTime_s < 0.0)
	OR (AR_Param.LS1.ConfirmTime_s > AR_Constant.CONFIRM_TIME_MAX_S) THEN
	AR_Internal.ConfigValid := FALSE;
	AR_Internal.ConfigFaultText := 'LS1 ConfirmTime_s mora biti 0..3600 s';
ELSIF (AR_Param.NumberOfLS >= 2)
	AND ((AR_Param.LS2.SP_Percent < AR_Constant.PCT_MIN)
		OR (AR_Param.LS2.SP_Percent > AR_Constant.PCT_MAX)) THEN
	AR_Internal.ConfigValid := FALSE;
	AR_Internal.ConfigFaultText := 'LS2 SP mora biti u opsegu 0..100%';
ELSIF (AR_Param.NumberOfLS >= 2)
	AND (AR_Param.LS2.Ramp_PercentPerSecond < AR_Constant.RAMP_MIN) THEN
	AR_Internal.ConfigValid := FALSE;
	AR_Internal.ConfigFaultText := 'LS2 rampa mora biti veca od 0%/s';
ELSIF (AR_Param.NumberOfLS >= 2)
	AND ((AR_Param.LS2.ConfirmTime_s < 0.0)
		OR (AR_Param.LS2.ConfirmTime_s > AR_Constant.CONFIRM_TIME_MAX_S)) THEN
	AR_Internal.ConfigValid := FALSE;
	AR_Internal.ConfigFaultText := 'LS2 ConfirmTime_s mora biti 0..3600 s';
ELSIF (AR_Param.NumberOfLS >= 2)
	AND (AR_Param.LS2.SP_Percent < AR_Param.LS1.SP_Percent) THEN
	AR_Internal.ConfigValid := FALSE;
	AR_Internal.ConfigFaultText := 'LS2 SP mora biti veci ili jednak LS1 SP';
ELSIF (AR_Param.NumberOfLS = 3)
	AND ((AR_Param.LS3.SP_Percent < AR_Constant.PCT_MIN)
		OR (AR_Param.LS3.SP_Percent > AR_Constant.PCT_MAX)) THEN
	AR_Internal.ConfigValid := FALSE;
	AR_Internal.ConfigFaultText := 'LS3 SP mora biti u opsegu 0..100%';
ELSIF (AR_Param.NumberOfLS = 3)
	AND (AR_Param.LS3.Ramp_PercentPerSecond < AR_Constant.RAMP_MIN) THEN
	AR_Internal.ConfigValid := FALSE;
	AR_Internal.ConfigFaultText := 'LS3 rampa mora biti veca od 0%/s';
ELSIF (AR_Param.NumberOfLS = 3)
	AND ((AR_Param.LS3.ConfirmTime_s < 0.0)
		OR (AR_Param.LS3.ConfirmTime_s > AR_Constant.CONFIRM_TIME_MAX_S)) THEN
	AR_Internal.ConfigValid := FALSE;
	AR_Internal.ConfigFaultText := 'LS3 ConfirmTime_s mora biti 0..3600 s';
ELSIF (AR_Param.NumberOfLS = 3)
	AND (AR_Param.LS3.SP_Percent < AR_Param.LS2.SP_Percent) THEN
	AR_Internal.ConfigValid := FALSE;
	AR_Internal.ConfigFaultText := 'LS3 SP mora biti veci ili jednak LS2 SP';
END_IF;

IF AR_Internal.ConfigValid THEN
	AR_Internal.LS1ConfirmTime := REAL_TO_TIME(AR_Param.LS1.ConfirmTime_s * 1000.0);
	AR_Internal.LS2ConfirmTime := REAL_TO_TIME(AR_Param.LS2.ConfirmTime_s * 1000.0);
	AR_Internal.LS3ConfirmTime := REAL_TO_TIME(AR_Param.LS3.ConfirmTime_s * 1000.0);
ELSE
	AR_Internal.LS1ConfirmTime := T#1s;
	AR_Internal.LS2ConfirmTime := T#1s;
	AR_Internal.LS3ConfirmTime := T#1s;
END_IF;

(* -------------------------------------------------------------------------- *)
(* 3) Dvosmerna vremenska potvrda LS signala                                  *)
(* -------------------------------------------------------------------------- *)
AR_Internal.TonLS1Change.IN :=
	AR_Internal.ConfigValid
	AND (AR_Input.LS1_Upper <> AR_Internal.LS1Confirmed);
AR_Internal.TonLS1Change.PT := AR_Internal.LS1ConfirmTime;
AR_Internal.TonLS1Change();

IF AR_Internal.TonLS1Change.Q THEN
	AR_Internal.LS1Confirmed := AR_Input.LS1_Upper;
END_IF;

IF AR_Param.NumberOfLS >= 2 THEN
	AR_Internal.TonLS2Change.IN :=
		AR_Internal.ConfigValid
		AND (AR_Input.LS2_Middle <> AR_Internal.LS2Confirmed);
	AR_Internal.TonLS2Change.PT := AR_Internal.LS2ConfirmTime;
	AR_Internal.TonLS2Change();

	IF AR_Internal.TonLS2Change.Q THEN
		AR_Internal.LS2Confirmed := AR_Input.LS2_Middle;
	END_IF;
ELSE
	AR_Internal.TonLS2Change(IN := FALSE, PT := T#0ms);
	AR_Internal.LS2Confirmed := FALSE;
END_IF;

IF AR_Param.NumberOfLS = 3 THEN
	AR_Internal.TonLS3Change.IN :=
		AR_Internal.ConfigValid
		AND (AR_Input.LS3_Lower <> AR_Internal.LS3Confirmed);
	AR_Internal.TonLS3Change.PT := AR_Internal.LS3ConfirmTime;
	AR_Internal.TonLS3Change();

	IF AR_Internal.TonLS3Change.Q THEN
		AR_Internal.LS3Confirmed := AR_Input.LS3_Lower;
	END_IF;
ELSE
	AR_Internal.TonLS3Change(IN := FALSE, PT := T#0ms);
	AR_Internal.LS3Confirmed := FALSE;
END_IF;

(* -------------------------------------------------------------------------- *)
(* 4) Monitoring aktivnog pritiska sa histerezom                              *)
(* -------------------------------------------------------------------------- *)
IF NOT AR_Input.Enable OR NOT AR_Internal.ConfigValid THEN
	AR_Internal.PressureActive := FALSE;
ELSIF NOT AR_Internal.PressureActive THEN
	IF AR_Input.Pressure_bar > AR_Param.PressureSP_bar THEN
		AR_Internal.PressureActive := TRUE;
	END_IF;
ELSIF AR_Input.Pressure_bar <
	(AR_Param.PressureSP_bar - AR_Param.PressureHysteresis_bar) THEN
	AR_Internal.PressureActive := FALSE;
END_IF;

(* -------------------------------------------------------------------------- *)
(* 5) Validacija fizickog redosleda potvrdenih LS signala                     *)
(* -------------------------------------------------------------------------- *)
AR_Internal.LSSequenceInvalid := FALSE;

IF AR_Internal.ConfigValid THEN
	CASE AR_Param.NumberOfLS OF
		2:
			AR_Internal.LSSequenceInvalid :=
				AR_Internal.LS1Confirmed
				AND NOT AR_Internal.LS2Confirmed;
		3:
			AR_Internal.LSSequenceInvalid :=
				(AR_Internal.LS1Confirmed AND NOT AR_Internal.LS2Confirmed)
				OR (AR_Internal.LS2Confirmed AND NOT AR_Internal.LS3Confirmed);
	END_CASE;
END_IF;

(* -------------------------------------------------------------------------- *)
(* 6) Aktivni alarmni uslov, latch i kontrolisani reset                       *)
(* -------------------------------------------------------------------------- *)
AR_Internal.ActiveConditionCode := AR_Constant.ACT_NONE;

IF NOT AR_Internal.ConfigValid THEN
	AR_Internal.ActiveConditionCode := AR_Constant.ACT_CONFIG_INVALID;
ELSIF NOT AR_Internal.RuntimeTimeValid THEN
	AR_Internal.ActiveConditionCode := AR_Constant.ACT_RUNTIME_TIME_INVALID;
ELSIF AR_Internal.LSSequenceInvalid THEN
	AR_Internal.ActiveConditionCode := AR_Constant.ACT_LS_SEQUENCE_INVALID;
END_IF;

AR_Internal.FaultCondition :=
	AR_Internal.ActiveConditionCode <> AR_Constant.ACT_NONE;

IF AR_Internal.FaultCondition THEN
	IF NOT AR_Internal.FaultLatched THEN
		CASE AR_Internal.ActiveConditionCode OF
			1: AR_Internal.FaultCode := AR_Constant.FLT_CONFIG_INVALID;
			2: AR_Internal.FaultCode := AR_Constant.FLT_LS_SEQUENCE_INVALID;
			3: AR_Internal.FaultCode := AR_Constant.FLT_RUNTIME_TIME_INVALID;
		ELSE
			AR_Internal.FaultCode := AR_Constant.FLT_NONE;
		END_CASE;
	END_IF;
	AR_Internal.FaultLatched := TRUE;
END_IF;

AR_Internal.ResetAllowed :=
	AR_Internal.FaultLatched
	AND NOT AR_Internal.FaultCondition
	AND AR_Internal.ConfigValid
	AND AR_Internal.RuntimeTimeValid;

IF AR_Input.ResetAlarm AND AR_Internal.ResetAllowed THEN
	AR_Internal.FaultLatched := FALSE;
	AR_Internal.FaultCode := AR_Constant.FLT_NONE;
END_IF;

(* -------------------------------------------------------------------------- *)
(* 7) Izbor manual komande ili automatskog LS stepena                         *)
(* -------------------------------------------------------------------------- *)
IF NOT AR_Input.Enable
	OR (NOT AR_Internal.PressureActive AND NOT AR_Input.EnableManual)
	OR AR_Internal.FaultCondition
	OR AR_Internal.FaultLatched THEN
	(* Bez dozvole, pritiska ili pri alarmu: isto kao potvrden gornji LS1. *)
	AR_Internal.OpeningMode := FALSE;
	AR_Internal.ActiveStage := 1;
	IF AR_Internal.ConfigValid THEN
		IF AR_Internal.ValveCmd > AR_Param.LS1.SP_Percent THEN
			AR_Internal.ValveCmd := AR_Param.LS1.SP_Percent;
		END_IF;
	ELSIF AR_Internal.ValveCmd > AR_Constant.SAFE_CLOSE_SP THEN
		AR_Internal.ValveCmd := AR_Constant.SAFE_CLOSE_SP;
	END_IF;
ELSIF AR_Input.EnableManual THEN
	(* Manual ima prioritet nad pressure/LS automatikom, ali ne nad Enable/fault. *)
	AR_Internal.ActiveStage := 0;
	AR_Internal.OpeningMode := FALSE;
	IF AR_Input.ManualSP_Percent < AR_Constant.PCT_MIN THEN
		AR_Internal.ValveCmd := AR_Constant.PCT_MIN;
	ELSIF AR_Input.ManualSP_Percent > AR_Constant.PCT_MAX THEN
		AR_Internal.ValveCmd := AR_Constant.PCT_MAX;
	ELSE
		AR_Internal.ValveCmd := AR_Input.ManualSP_Percent;
	END_IF;
ELSIF NOT AR_Internal.ControlActivePrev THEN
	(* Prvi aktivni scan bira stanje prema najvisem potvrdenom LS-u. *)
	IF AR_Internal.LS1Confirmed THEN
		AR_Internal.OpeningMode := FALSE;
		AR_Internal.ActiveStage := 1;
		IF AR_Internal.ValveCmd > AR_Param.LS1.SP_Percent THEN
			AR_Internal.ValveCmd := AR_Param.LS1.SP_Percent;
		END_IF;
	ELSIF (AR_Param.NumberOfLS >= 2) AND AR_Internal.LS2Confirmed THEN
		AR_Internal.OpeningMode := FALSE;
		AR_Internal.ActiveStage := 1;
		IF AR_Internal.ValveCmd > AR_Param.LS1.SP_Percent THEN
			AR_Internal.ValveCmd := AR_Param.LS1.SP_Percent;
		END_IF;
	ELSIF (AR_Param.NumberOfLS = 3) AND AR_Internal.LS3Confirmed THEN
		AR_Internal.OpeningMode := FALSE;
		AR_Internal.ActiveStage := 2;
		IF AR_Internal.ValveCmd > AR_Param.LS2.SP_Percent THEN
			AR_Internal.ValveCmd := AR_Param.LS2.SP_Percent;
		END_IF;
	ELSE
		AR_Internal.OpeningMode := TRUE;
		AR_Internal.ActiveStage := AR_Param.NumberOfLS;
	END_IF;
ELSE
	(* Aktivacija vode ima prioritet; najvisi novi LS odreduje trenutni clamp. *)
	IF AR_Internal.LS1Confirmed AND NOT AR_Internal.LS1ConfirmedPrev THEN
		AR_Internal.OpeningMode := FALSE;
		AR_Internal.ActiveStage := 1;
		IF AR_Internal.ValveCmd > AR_Param.LS1.SP_Percent THEN
			AR_Internal.ValveCmd := AR_Param.LS1.SP_Percent;
		END_IF;
	ELSIF (AR_Param.NumberOfLS >= 2)
		AND AR_Internal.LS2Confirmed
		AND NOT AR_Internal.LS2ConfirmedPrev THEN
		AR_Internal.OpeningMode := FALSE;
		AR_Internal.ActiveStage := 1;
		IF AR_Internal.ValveCmd > AR_Param.LS1.SP_Percent THEN
			AR_Internal.ValveCmd := AR_Param.LS1.SP_Percent;
		END_IF;
	ELSIF (AR_Param.NumberOfLS = 3)
		AND AR_Internal.LS3Confirmed
		AND NOT AR_Internal.LS3ConfirmedPrev THEN
		AR_Internal.OpeningMode := FALSE;
		AR_Internal.ActiveStage := 2;
		IF AR_Internal.ValveCmd > AR_Param.LS2.SP_Percent THEN
			AR_Internal.ValveCmd := AR_Param.LS2.SP_Percent;
		END_IF;
	ELSIF (AR_Param.NumberOfLS = 3)
		AND NOT AR_Internal.LS3Confirmed
		AND AR_Internal.LS3ConfirmedPrev THEN
		AR_Internal.OpeningMode := TRUE;
		AR_Internal.ActiveStage := 3;
	ELSIF (AR_Param.NumberOfLS >= 2)
		AND NOT AR_Internal.LS2Confirmed
		AND AR_Internal.LS2ConfirmedPrev THEN
		AR_Internal.OpeningMode := TRUE;
		AR_Internal.ActiveStage := 2;
	ELSIF NOT AR_Internal.LS1Confirmed
		AND AR_Internal.LS1ConfirmedPrev THEN
		AR_Internal.OpeningMode := TRUE;
		AR_Internal.ActiveStage := 1;
	END_IF;
END_IF;

(* -------------------------------------------------------------------------- *)
(* 8) Izbor cilja i rampe automatskog stepena                                *)
(* -------------------------------------------------------------------------- *)
IF AR_Input.EnableManual
	AND AR_Input.Enable
	AND NOT AR_Internal.FaultCondition
	AND NOT AR_Internal.FaultLatched THEN
	AR_Internal.TargetSP := AR_Internal.ValveCmd;
	AR_Internal.ActiveRamp := 0.0;
ELSE
	CASE AR_Internal.ActiveStage OF
		1:
			IF AR_Internal.ConfigValid THEN
				AR_Internal.ActiveRamp := AR_Param.LS1.Ramp_PercentPerSecond;
			ELSE
				AR_Internal.ActiveRamp := AR_Constant.SAFE_CLOSE_RAMP;
			END_IF;
			IF AR_Internal.OpeningMode AND AR_Internal.ConfigValid THEN
				AR_Internal.TargetSP := AR_Param.LS1.SP_Percent;
			ELSE
				AR_Internal.TargetSP := AR_Constant.PCT_MIN;
			END_IF;
		2:
			AR_Internal.ActiveRamp := AR_Param.LS2.Ramp_PercentPerSecond;
			IF AR_Internal.OpeningMode THEN
				AR_Internal.TargetSP := AR_Param.LS2.SP_Percent;
			ELSE
				AR_Internal.TargetSP := AR_Constant.PCT_MIN;
			END_IF;
		3:
			AR_Internal.ActiveRamp := AR_Param.LS3.Ramp_PercentPerSecond;
			IF AR_Internal.OpeningMode THEN
				AR_Internal.TargetSP := AR_Param.LS3.SP_Percent;
			ELSE
				AR_Internal.TargetSP := AR_Constant.PCT_MIN;
			END_IF;
	ELSE
		AR_Internal.ActiveStage := 1;
		AR_Internal.ActiveRamp := AR_Param.LS1.Ramp_PercentPerSecond;
		AR_Internal.TargetSP := AR_Constant.PCT_MIN;
	END_CASE;
END_IF;

(* -------------------------------------------------------------------------- *)
(* 9) Rampa komande u %/s prema stvarnom vremenu task ciklusa                 *)
(* -------------------------------------------------------------------------- *)
IF AR_Input.EnableManual
	AND AR_Input.Enable
	AND NOT AR_Internal.FaultCondition
	AND NOT AR_Internal.FaultLatched THEN
	(* Direktna manual komanda ne koristi procesnu rampu. *)
ELSIF AR_Internal.RuntimeTimeValid THEN
	AR_Internal.RampStep := AR_Internal.ActiveRamp * AR_Output.CycleTime_s;

	IF AR_Internal.TargetSP > AR_Internal.ValveCmd THEN
		AR_Internal.ValveCmd := AR_Internal.ValveCmd + AR_Internal.RampStep;
		IF AR_Internal.ValveCmd > AR_Internal.TargetSP THEN
			AR_Internal.ValveCmd := AR_Internal.TargetSP;
		END_IF;
	ELSIF AR_Internal.TargetSP < AR_Internal.ValveCmd THEN
		AR_Internal.ValveCmd := AR_Internal.ValveCmd - AR_Internal.RampStep;
		IF AR_Internal.ValveCmd < AR_Internal.TargetSP THEN
			AR_Internal.ValveCmd := AR_Internal.TargetSP;
		END_IF;
	END_IF;
ELSIF AR_Internal.FaultCondition THEN
	(* Bez validne vremenske baze nije moguca kontrolisana rampa. *)
	AR_Internal.ValveCmd := AR_Constant.PCT_MIN;
END_IF;

IF AR_Internal.ValveCmd < AR_Constant.PCT_MIN THEN
	AR_Internal.ValveCmd := AR_Constant.PCT_MIN;
ELSIF AR_Internal.ValveCmd > AR_Constant.PCT_MAX THEN
	AR_Internal.ValveCmd := AR_Constant.PCT_MAX;
END_IF;

(* -------------------------------------------------------------------------- *)
(* 10) State, tekst i HMI dijagnostika                                        *)
(* -------------------------------------------------------------------------- *)
IF AR_Internal.FaultCondition OR AR_Internal.FaultLatched THEN
	AR_Internal.Step := AR_Constant.ST_FAULT_SAFE_CLOSE;
ELSIF NOT AR_Input.Enable THEN
	AR_Internal.Step := AR_Constant.ST_DISABLED;
ELSIF AR_Input.EnableManual THEN
	AR_Internal.Step := AR_Constant.ST_MANUAL;
ELSIF NOT AR_Internal.PressureActive THEN
	AR_Internal.Step := AR_Constant.ST_WAIT_PRESSURE;
ELSIF AR_Internal.ValveCmd <= AR_Constant.PCT_MIN THEN
	AR_Internal.Step := AR_Constant.ST_CLOSED;
ELSIF AR_Internal.OpeningMode THEN
	CASE AR_Internal.ActiveStage OF
		1: AR_Internal.Step := AR_Constant.ST_OPENING_LS1;
		2: AR_Internal.Step := AR_Constant.ST_OPENING_LS2;
		3: AR_Internal.Step := AR_Constant.ST_OPENING_LS3;
	END_CASE;
ELSE
	CASE AR_Internal.ActiveStage OF
		1: AR_Internal.Step := AR_Constant.ST_CLOSING_LS1;
		2: AR_Internal.Step := AR_Constant.ST_CLOSING_LS2;
	ELSE
		AR_Internal.Step := AR_Constant.ST_CLOSING_LS1;
	END_CASE;
END_IF;

CASE AR_Internal.Step OF
	0: AR_Output.State_comment := 'ST_DISABLED - bezbedno zatvaranje ventila';
	1: AR_Output.State_comment := 'ST_WAIT_PRESSURE - ceka aktivni pritisak';
	2: AR_Output.State_comment := 'ST_OPENING_LS1 - otvaranje rampom LS1';
	3: AR_Output.State_comment := 'ST_OPENING_LS2 - otvaranje rampom LS2';
	4: AR_Output.State_comment := 'ST_OPENING_LS3 - otvaranje rampom LS3';
	5: AR_Output.State_comment := 'ST_CLOSING_LS1 - zatvaranje rampom LS1';
	6: AR_Output.State_comment := 'ST_CLOSING_LS2 - zatvaranje rampom LS2';
	7: AR_Output.State_comment := 'ST_CLOSED - komanda ventila je 0%';
	8: AR_Output.State_comment := 'ST_FAULT_SAFE_CLOSE - alarm, bezbedno zatvaranje';
	9: AR_Output.State_comment := 'ST_MANUAL - direktna rucna komanda 0..100%';
ELSE
	AR_Output.State_comment := 'ST_UNKNOWN - nepoznato stanje';
END_CASE;

CASE AR_Internal.FaultCode OF
	0: AR_Output.FaultText := 'FLT_NONE - nema memorisanog alarma';
	1: AR_Output.FaultText := 'FLT_CONFIG_INVALID - nevalidni parametri';
	2: AR_Output.FaultText := 'FLT_LS_SEQUENCE_INVALID - nelogican LS redosled';
	3: AR_Output.FaultText := 'FLT_RUNTIME_TIME_INVALID - nema vremena ciklusa';
ELSE
	AR_Output.FaultText := 'FLT_UNKNOWN - nepoznat memorisani alarm';
END_CASE;

IF NOT AR_Internal.ConfigValid THEN
	AR_Output.Diag := 'CONFIG_INVALID';
ELSIF NOT AR_Internal.RuntimeTimeValid THEN
	AR_Output.Diag := 'RUNTIME_TIME_INVALID';
ELSIF AR_Internal.LSSequenceInvalid THEN
	AR_Output.Diag := 'LS_SEQUENCE_INVALID';
ELSIF AR_Internal.FaultLatched THEN
	AR_Output.Diag := 'ALARM_LATCHED_WAIT_RESET';
ELSIF NOT AR_Input.Enable THEN
	AR_Output.Diag := 'DISABLED_SAFE_CLOSING';
ELSIF AR_Input.EnableManual THEN
	AR_Output.Diag := 'MANUAL_DIRECT_COMMAND';
ELSIF NOT AR_Internal.PressureActive THEN
	AR_Output.Diag := 'WAITING_ACTIVE_PRESSURE';
ELSIF AR_Internal.OpeningMode THEN
	AR_Output.Diag := 'AIR_RELEASE_OPENING';
ELSE
	AR_Output.Diag := 'WATER_CONFIRMED_CLOSING';
END_IF;

(* -------------------------------------------------------------------------- *)
(* 11) Izlazno mapiranje                                                       *)
(* -------------------------------------------------------------------------- *)
AR_Output.ValveSP_Percent := AR_Internal.ValveCmd;
AR_Output.Status :=
	AR_Input.Enable
	AND AR_Internal.ConfigValid
	AND AR_Internal.RuntimeTimeValid
	AND NOT AR_Internal.FaultLatched;
AR_Output.State := AR_Internal.Step;
AR_Output.ManualActive :=
	AR_Input.Enable
	AND AR_Input.EnableManual
	AND NOT AR_Internal.FaultCondition
	AND NOT AR_Internal.FaultLatched;
AR_Output.PressureActive := AR_Internal.PressureActive;
AR_Output.LS1_Confirmed := AR_Internal.LS1Confirmed;
AR_Output.LS2_Confirmed := AR_Internal.LS2Confirmed;
AR_Output.LS3_Confirmed := AR_Internal.LS3Confirmed;
AR_Output.ActiveStage := AR_Internal.ActiveStage;
AR_Output.Opening := NOT AR_Output.ManualActive
	AND AR_Internal.OpeningMode
	AND (AR_Internal.ValveCmd < AR_Internal.TargetSP);
AR_Output.Closing := NOT AR_Output.ManualActive
	AND NOT AR_Internal.OpeningMode
	AND (AR_Internal.ValveCmd > AR_Constant.PCT_MIN);
AR_Output.AlarmActive := AR_Internal.FaultCondition;
AR_Output.AlarmLatched := AR_Internal.FaultLatched;
AR_Output.FaultCode := AR_Internal.FaultCode;
AR_Output.ActiveConditionCode := AR_Internal.ActiveConditionCode;
AR_Output.ResetAllowed := AR_Internal.ResetAllowed;
AR_Output.ConfigValid := AR_Internal.ConfigValid;
AR_Output.ConfigFaultText := AR_Internal.ConfigFaultText;
AR_Output.LSSequenceInvalid := AR_Internal.LSSequenceInvalid;

(* -------------------------------------------------------------------------- *)
(* 12) Memorija prethodnog ciklusa                                            *)
(* -------------------------------------------------------------------------- *)
AR_Internal.ControlActivePrev :=
	AR_Input.Enable
	AND NOT AR_Input.EnableManual
	AND AR_Internal.PressureActive
	AND NOT AR_Internal.FaultCondition
	AND NOT AR_Internal.FaultLatched;
AR_Internal.LS1ConfirmedPrev := AR_Internal.LS1Confirmed;
AR_Internal.LS2ConfirmedPrev := AR_Internal.LS2Confirmed;
AR_Internal.LS3ConfirmedPrev := AR_Internal.LS3Confirmed;

END_FUNCTION_BLOCK
```

### Library Logical/Libraries/VFD_Lib (IEC, version 6.03.0)

#### Types.typ - Exported data types
```iecst
TYPE
	(* ======================================================================== *)
	(* Glavni agregatni tip za VFD instancu                                    *)
	(* ======================================================================== *)
	VFD_type : 	STRUCT (* Glavna agregatna struktura jedne VFD instance. *)
		cmds : vfd_commands;              (* Komandni zahtevi ka frekventnom regulatoru – sve upravljačke komande za VFD instancu. *)
		params : vfd_set_parameters;      (* Procesni setpoint-i i dinamika (acc/dec) – parametri zadavanja brzine, ubrzanja i usporenja. *)
		mapping : vfd_mapping;            (* Niskonivo mapiranje I/O i fieldbus registara – fizičko/logičko mapiranje signala. *)
		states : vfd_states;              (* Dekodirana operativna stanja regulatora – statusni bitovi i stanja rada. *)
		status : vfd_status;              (* Aktuelne merene vrednosti regulatora/motora – procesni izlazi. *)
		errorID : UINT;                   (* Numerički kod greške iz komunikacije/drive-a – za dijagnostiku. *)
		errorText : STRING[40];           (* Kratak tekstualni opis greške za HMI – olakšava korisničku dijagnostiku. *)
		settings : vfd_settings_param;    (* Konfiguracija metode rada i granica – podešavanja instance. *)
		errorMgmt : vfd_errorMgmt;        (* Statistika i trajanje prekida komunikacije – monitoring pouzdanosti. *)
	END_STRUCT;

	(* ======================================================================== *)
	(* Procesni status izlazi                                                   *)
	(* ======================================================================== *)
	vfd_status : 	STRUCT (* Procesni status izlaza – merene vrednosti pogona. *)
		act_velocity : REAL;      (* Trenutna brzina motora [r/min]. *)
		act_power : REAL;         (* Trenutna snaga motora [kW]. *)
		act_torque : REAL;        (* Trenutni obrtni moment [Nm] – zavisi od mapiranja drive-a. *)
		act_voltage : REAL;       (* Trenutni napon motora [V]. *)
		act_freq : REAL;          (* Trenutna frekvencija izlaza [Hz]. *)
		act_current : REAL;       (* Trenutna struja motora [A]. *)
	END_STRUCT;

	(* ======================================================================== *)
	(* Dekodirana stanja rada VFD                                               *)
	(* ======================================================================== *)
	vfd_states : 	STRUCT (* Dekodirana radna stanja VFD-a i statusni bitovi. *)
		PWR_ON : BOOL := FALSE;              (* Napajanje/drive aktivan – glavni naponski izvor uključen. *)
		ALARM : BOOL := FALSE;               (* Alarm stanje bez hard fault latch-a – signalizacija upozorenja. *)
		FAULT : BOOL := FALSE;               (* Fault stanje regulatora – kritična greška, rad onemogućen. *)
		TUNING : BOOL := FALSE;              (* Aktivno tuning/samopodešavanje – automatska optimizacija parametara. *)
		READY : BOOL := FALSE;               (* Drive spreman za komandu rada – svi uslovi za start su ispunjeni. *)
		PREOPERATIONAL : BOOL := FALSE;      (* Pre-run tranziciono stanje – prelazna faza pre rada. *)
		JOG : BOOL := FALSE;                 (* Jog režim aktivan – ručno pokretanje za podešavanje. *)
		RUN : BOOL := FALSE;                 (* Kontinualni rad aktivan – normalan režim pogona. *)
		STOPPING : BOOL := FALSE;            (* U toku kontrolisano zaustavljanje – sekvenca zaustavljanja. *)
		STOPED : BOOL := FALSE;              (* Zaustavljen (zadržan originalni naziv) – pogon je stao. *)
		OVERCURRENT_PROTECT : BOOL := FALSE; (* Aktivna zaštita od prekostruje – zaštitna funkcija. *)
		state_word : UINT := 0;              (* Sirovi/dekodirani state kod za internu obradu – za naprednu dijagnostiku. *)
	END_STRUCT;

	(* ======================================================================== *)
	(* Parametri setovanja                                                       *)
	(* ======================================================================== *)
	vfd_set_parameters : 	STRUCT (* Parametri zadavanja brzine i dinamike pogona. *)
		Freq : REAL;         (* Glavna zadavana frekvencija [Hz] – opseg 0–100.00. *)
		Jog_freq : REAL;     (* Posebna jog frekvencija [Hz] – za ručno pokretanje. *)
		Dec : REAL;          (* Vreme/uslov usporavanja [s] – prema mapiranju drive-a. *)
		Acc : REAL;          (* Vreme/uslov ubrzavanja [s] – prema mapiranju drive-a. *)
	END_STRUCT;

	(* ======================================================================== *)
	(* Grupisano mapiranje po metodi upravljanja                                *)
	(* ======================================================================== *)
	vfd_mapping : 	STRUCT (* Grupisano mapiranje signala po metodi upravljanja. *)
		DIO : vfd_maping_DIO;              (* Diskretno/analogno mapiranje preko I/O signala – osnovni digitalni/analogni signali. *)
		CanOpenATV : vfd_maping_CanOpenATV;(* CANopen mapiranje za ATV varijantu – komunikacija sa ATV uređajem. *)
		CanOpen : vfd_maping_CanOpenENC;   (* CANopen mapiranje za ENC varijantu – komunikacija sa ENC uređajem. *)
	END_STRUCT;

	(* ======================================================================== *)
	(* DIO mapiranje                                                             *)
	(* ======================================================================== *)
	vfd_maping_DIO : 	STRUCT (* DIO mapiranje komandi i povratnih signala. *)
		w_run_fwd : BOOL;         (* Komanda: rad napred – pokretanje motora unapred. *)
		w_run_rev : BOOL;         (* Komanda: rad nazad – pokretanje motora unazad. *)
		w_jog_fwd : BOOL;         (* Komanda: jog napred – ručno pokretanje unapred. *)
		w_jog_rev : BOOL;         (* Komanda: jog nazad – ručno pokretanje unazad. *)
		w_Stop : BOOL;            (* Komanda: standard stop – normalno zaustavljanje. *)
		w_faststop : BOOL;        (* Komanda: brzi stop – hitno zaustavljanje. *)
		w_reset : BOOL;           (* Komanda: reset greške – resetuje fault/grešku. *)
		w_freq : INT;             (* Upisana frekvencija/komanda (raw) – zadavanje brzine. *)
		r_freq : INT;             (* Pročitana frekvencija (raw) – povratna informacija. *)
		r_OverCurrentProtect : BOOL; (* Povratni signal zaštite od prekostruje – signalizacija zaštite. *)
		r_error : BOOL;           (* Povratni signal opšte greške drive-a – signalizacija kvara. *)
	END_STRUCT;

	(* ======================================================================== *)
	(* CANopen ATV mapiranje                                                     *)
	(* ======================================================================== *)
	vfd_maping_CanOpenATV : 	STRUCT (* CANopen mapiranje za ATV varijantu pogona. *)
		StatusWord : UINT;            (* Status reč sa CANopen uređaja – statusni bitovi pogona. *)
		CtrlWord : UINT;              (* Komandna reč ka CANopen uređaju – upravljački zahtevi. *)
		r_freq : INT;                 (* Pročitana frekvencija (raw skala ATV) – povratna vrednost. *)
		r_power : INT;                (* Pročitana snaga (raw/procenat, zavisi od mapiranja). *)
		r_current : UINT;             (* Pročitana struja (raw) – trenutna potrošnja. *)
		r_torque : INT;               (* Pročitani moment (raw) – trenutni obrtni moment. *)
		r_voltage : UINT;             (* Pročitan napon (raw) – trenutni napon. *)
		r_velocity : INT;             (* Pročitana brzina (raw) – trenutna brzina. *)
		r_CtrlWord : UINT;            (* Echo/feedback komandne reči – povratna informacija. *)
		r_errorCode : UINT;           (* Kod greške prijavljen od drive-a – dijagnostika. *)
		r_RatedMotorPower : UINT;     (* Nominalna snaga motora pročitana iz drive-a. *)
		r_OverCurrentProtect : BOOL;  (* Povratni signal overcurrent zaštite – signalizacija zaštite. *)
		w_TargetVelocity : INT;       (* Upis target brzine – zadavanje željene brzine. *)
		w_acc : UINT;                 (* Upis parametra acc – zadavanje ubrzanja. *)
		w_dec : UINT;                 (* Upis parametra dec – zadavanje usporenja. *)
		ControlEffort : INT;          (* Interni/eksterni effort signal (mapiran) – napor kontrole. *)
		ModuleStatusOK : BOOL;        (* Status komunikacionog modula za ATV kanal – TRUE=modul OK. *)
	END_STRUCT;

	(* ======================================================================== *)
	(* CANopen ENC mapiranje                                                     *)
	(* ======================================================================== *)
	vfd_maping_CanOpenENC : 	STRUCT (* CANopen mapiranje za ENC varijantu pogona. *)
		StatusWord : UINT;            (* Status reč sa CANopen uređaja – statusni bitovi pogona. *)
		CtrlWord : UINT;              (* Komandna reč ka CANopen uređaju – upravljački zahtevi. *)
		r_freq : UINT;                (* Pročitana frekvencija (raw) – povratna vrednost. *)
		r_power : UINT;               (* Pročitana snaga (raw) – trenutna snaga. *)
		r_current : UINT;             (* Pročitana struja (raw) – trenutna potrošnja. *)
		r_torque : UINT;              (* Pročitani moment (raw) – trenutni obrtni moment. *)
		r_voltage : UINT;             (* Pročitan napon (raw) – trenutni napon. *)
		r_velocity : UINT;            (* Pročitana brzina (raw) – trenutna brzina. *)
		r_CtrlWord : UINT;            (* Echo/feedback komandne reči – povratna informacija. *)
		r_errorCode : UINT;           (* Kod greške prijavljen od drive-a – dijagnostika. *)
		r_OverCurrentProtect : BOOL;  (* Povratni signal overcurrent zaštite – signalizacija zaštite. *)
		w_acc : UINT;                 (* Upis parametra acc – zadavanje ubrzanja. *)
		w_dec : UINT;                 (* Upis parametra dec – zadavanje usporenja. *)
		w_freq : UINT;                (* Upis komandne frekvencije (raw) – zadavanje brzine. *)
		ModuleStatusOK : BOOL;        (* Status komunikacionog modula za ENC kanal – TRUE=modul OK. *)
	END_STRUCT;

	(* ======================================================================== *)
	(* Upravljanje greskama komunikacije                                         *)
	(* ======================================================================== *)
	vfd_errorMgmt : 	STRUCT (* Evidencija i status prekida komunikacije. *)
		Last_time : DATE_AND_TIME;    (* Vreme poslednjeg završenog komunikacionog ispada – za istoriju. *)
		Last_Duration : TIME;         (* Trajanje poslednjeg ispada [ms]. *)
		Counter_errors : DINT;        (* Broj registrovanih prekida komunikacije – ukupno. *)
		Max_duration : TIME;          (* Najduže trajanje pojedinačnog prekida [ms]. *)
		StatusOK : BOOL;              (* Trenutni status komunikacije (TRUE=OK). *)
	END_STRUCT;

	(* ======================================================================== *)
	(* Parametri konfiguracije instance                                           *)
	(* ======================================================================== *)
	vfd_settings_param : 	STRUCT (* Konfiguracioni parametri rada i granice instance. *)
		METOD_OF_CONTROL : USINT;         (* Izabrani metod upravljanja (DIO/CANopen varijante) – način kontrole. *)
		MIN_Freq : REAL;                  (* Minimalna dozvoljena frekvencija [Hz]. *)
		MAX_Freq : REAL;                  (* Maksimalna dozvoljena frekvencija [Hz]. *)
		MAX_Velocity : REAL;              (* Maksimalna brzina motora [r/min]. *)
		RatedMotorPower : REAL;           (* Nominalna snaga motora sa natpisne pločice [kW]. *)
		HaveOverCurrentProtection : BOOL; (* TRUE=ima zaštitu od prekostruje, FALSE=nema. *)
	END_STRUCT;

	(* ======================================================================== *)
	(* Komande upravljanja                                                       *)
	(* ======================================================================== *)
	vfd_commands : 	STRUCT (* Upravljačke komande za rad VFD instance. *)
		Enable : BOOL;                (* Glavni enable bloka i komandi – omogućava rad instance. *)
		FastStop : BOOL;              (* Prioritetna komanda brzog zaustavljanja – hitno zaustavljanje. *)
		Stop : BOOL;                  (* Standardna stop komanda – normalno zaustavljanje. *)
		Run_fwd : BOOL;               (* Kontinualni rad napred – pokretanje motora unapred. *)
		Run_rev : BOOL;               (* Kontinualni rad nazad – pokretanje motora unazad. *)
		Jog_rev : BOOL;               (* Jog nazad – ručno pokretanje unazad. *)
		Jog_fwd : BOOL;               (* Jog napred – ručno pokretanje unapred. *)
		en_autoReset : BOOL := TRUE;  (* Automatski reset odabranih fault uslova – automatsko otklanjanje grešaka. *)
		Reset : BOOL;                 (* Ručni reset fault/alarm stanja – manuelno otklanjanje grešaka. *)
	END_STRUCT;
END_TYPE
```

#### Constants.var - Exported constants
```iecst
VAR CONSTANT
	METOD_ATV_CANOPEN : USINT := 2; (* Metod upravljanja: ATV CANopen varijanta. *)
	METOD_DIO : USINT := 1; (* Metod upravljanja: diskretni/analogni I/O (DIO). *)
	METOD_DIO_CANOPEN : USINT := 3; (* Metod upravljanja: komande preko DIO, status preko CANopen. *)
	METOD_ENC_CANOPEN : USINT := 0; (* Metod upravljanja: ENC CANopen varijanta. *)
	STATV_ERR : USINT := 8; (* ATV stanje: greska (error). *)
	STATV_ERR_MNG : USINT := 7; (* ATV stanje: aktivan rezim upravljanja greskom. *)
	STATV_FAST_STOP : USINT := 6; (* ATV stanje: aktivno brzo zaustavljanje. *)
	STATV_OVR_CURR : USINT := 9; (* ATV stanje: aktivna zastita od prekostruje. *)
	STATV_PWR_OFF : USINT := 0; (* ATV stanje: pogon bez napajanja/iskljucen. *)
	STATV_RDY : USINT := 3; (* ATV stanje: spreman za start. *)
	STATV_RDY_NOT : USINT := 1; (* ATV stanje: nije spreman za start. *)
	STATV_RUN : USINT := 5; (* ATV stanje: pogon u radu (operation enabled). *)
	STATV_SWH_DISABLE : USINT := 2; (* ATV stanje: switch-on disabled. *)
	STATV_SWH_ON : USINT := 4; (* ATV stanje: switch-on aktivan. *)
	ST_ALARM : USINT := 7; (* Standardno stanje: alarm. *)
	ST_CURRPROTECT : USINT := 10; (* Standardno stanje: aktivna zastita od prekostruje. *)
	ST_FAULT : USINT := 6; (* Standardno stanje: greska. *)
	ST_JOG : USINT := 9; (* Standardno stanje: jog rezim. *)
	ST_PREOPERATIONAL : USINT := 2; (* Standardno stanje: prelazni rezim pre punog rada (ACC/DEC). *)
	ST_PWR_OFF : USINT := 0; (* Standardno stanje: bez napajanja/iskljucen. *)
	ST_READY : USINT := 1; (* Standardno stanje: spreman za rad. *)
	ST_RUN : USINT := 3; (* Standardno stanje: rad. *)
	ST_STOPPED : USINT := 5; (* Standardno stanje: zaustavljen. *)
	ST_STOPPING : USINT := 4; (* Standardno stanje: zaustavljanje u toku. *)
	ST_TUNING : USINT := 8; (* Standardno stanje: samopodesavanje aktivno. *)
END_VAR
```

#### VFD_Lib.fun - Exported functions and function blocks
```iecst
{REDUND_ERROR} FUNCTION_BLOCK fbCheckStateCanOpenENC (* Dekodiranje status reci CANopen ENC varijante u standardni state kod. *) (*$GROUP=User,$CAT=User,$GROUPICON=User.png,$CATICON=User.png*)
	VAR_INPUT (* Ulazni podaci za dekodiranje status reci. *)
		in_addr_StatusWord : {REDUND_UNREPLICABLE} UDINT; (* Adresa status reci uredjaja. *)
	END_VAR
	VAR_OUTPUT (* Izlaz dekodiranog internog state koda. *)
		out_State : UINT; (* Dekodirani interni state kod. *)
	END_VAR
	VAR (* Interne reference i pomocne promenljive bloka. *)
		ref_statusWord : REFERENCE TO UINT; (* Referenca na status rec zbog bit-level dekodiranja. *)
	END_VAR
END_FUNCTION_BLOCK

{REDUND_ERROR} FUNCTION_BLOCK fbControlCanOpenENC (* Komandovanje CANopen ENC varijante kroz CtrlWord sekvencu. *) (*$GROUP=User,$CAT=User,$GROUPICON=User.png,$CATICON=User.png*)
	VAR_INPUT (* Ulazni komandni i adresni podaci za ENC upravljanje. *)
		cmd : vfd_commands; (* Grupisane komande sa nadredjenog nivoa. *)
		in_addr_StatusWord : UDINT; (* Adresa status reci uredjaja. *)
		in_addr_r_CtrlWord : UDINT; (* Adresa povratne/eho komandne reci. *)
		in_addr_CtrlWord : UDINT; (* Adresa komandne reci za upis. *)
	END_VAR
	VAR_OUTPUT (* Izlazi statusa izvrsenja komandi. *)
		out_BUSY : BOOL; (* TRUE dok je tranzicija komande u toku. *)
		out_DONE : BOOL; (* TRUE kada je trazena komanda potvrdena. *)
	END_VAR
	VAR (* Interne reference i pomocni flagovi sekvence. *)
		en : BOOL; (* Interna kopija Enable logike. *)
		ref_statusWord : REFERENCE TO UINT; (* Referenca na status rec. *)
		r_ctrlWord : REFERENCE TO UINT; (* Referenca na feedback ctrl rec. *)
		ref_ctrlWord : REFERENCE TO UINT; (* Referenca na izlaznu ctrl rec. *)
		start_check : BOOL; (* Memorija za auto-reset sekvencu. *)
	END_VAR
END_FUNCTION_BLOCK

{REDUND_ERROR} FUNCTION_BLOCK vfdMain (* Glavni VFD blok: dispatch po metodi, kontrola i monitoring. *) (*$GROUP=User,$CAT=User,$GROUPICON=User.png,$CATICON=User.png*)
	VAR_INPUT (* Ulazni podaci instance glavnog VFD bloka. *)
		addr_struct : UDINT; (* Adresa agregatne VFD strukture (VFD_type). *)
	END_VAR
	VAR_OUTPUT (* Izlazni dijagnosticki i statusni signali bloka. *)
		errorID : UINT; (* Izlazni kod greske prema aktivnoj metodi mapiranja. *)
		errorText : STRING[40]; (* Izlazni tekst greske za HMI dijagnostiku. *)
		Done : BOOL; (* Operacija komande zavrsena. *)
		Busy : BOOL; (* Operacija komande je u toku. *)
	END_VAR
	VAR (* Interne FB instance, reference i pomocne promenljive. *)
		fControlENC : fbControlCanOpenENC; (* Komandni pod-blok za ENC varijantu. *)
		fStateENC : fbCheckStateCanOpenENC; (* State dekoder za ENC varijantu. *)
		fControlATV : fbControlCanOpenATV; (* Komandni pod-blok za ATV varijantu. *)
		fStateATV : fbCheckStateCanOpenATV; (* State dekoder za ATV varijantu. *)
		vfd_struct_data : REFERENCE TO VFD_type; (* Referenca ka centralnoj VFD strukturi. *)
		state_case : UINT; (* Privremeni state izbor za mapiranje izlaza states.*)
		acum_time : TIME; (* Akumulirano trajanje duzih prekida komunikacije. *)
		DTGetTime_1 : DTGetTime; (* Sistemski blok za uzimanje vremena dogadaja. *)
		ton_dur : TON; (* Tajmer trajanja komunikacionog ispada. *)
		zzEdge00000 : BOOL; (* Rezervisano/interne potrebe (legacy). *)
	END_VAR
END_FUNCTION_BLOCK

{REDUND_ERROR} FUNCTION_BLOCK fbCheckStateCanOpenATV (* Dekodiranje ATV status reci u ATV state kod. *) (*$GROUP=User,$CAT=User,$GROUPICON=User.png,$CATICON=User.png*)
	VAR_INPUT (* Ulazni podaci za dekodiranje ATV status reci. *)
		in_addr_StatusWord : {REDUND_UNREPLICABLE} UDINT; (* Adresa ATV status reci. *)
	END_VAR
	VAR_OUTPUT (* Izlaz dekodiranog ATV state koda i pomocnih stanja. *)
		out_State : {REDUND_UNREPLICABLE} UINT; (* Dekodirani ATV state kod. *)
		DC_BUS_ON : BOOL; (* Informacija da je DC bus aktivan. *)
	END_VAR
	VAR (* Interne reference za citanje status reci. *)
		ref_statusWord : REFERENCE TO UINT; (* Referenca na ATV status rec. *)
	END_VAR
END_FUNCTION_BLOCK

{REDUND_ERROR} FUNCTION_BLOCK fbControlCanOpenATV (* Komandovanje ATV CANopen varijante preko CtrlWord logike. *) (*$GROUP=User,$CAT=User,$GROUPICON=User.png,$CATICON=User.png*)
	VAR_INPUT (* Ulazni komandni i procesni podaci za ATV upravljanje. *)
		cmd : {REDUND_UNREPLICABLE} vfd_commands; (* Komande sa nadredjenog nivoa. *)
		in_set_freq : INT; (* Trazeni speed/freq setpoint u ATV skali. *)
		in_addr_CtrlWord : {REDUND_UNREPLICABLE} UDINT; (* Adresa ctrl reci za upis. *)
		StatusWord : {REDUND_UNREPLICABLE} UINT; (* Trenutni ATV state kod (dekodiran). *)
		DC_BUS_STATE : {REDUND_UNREPLICABLE} BOOL; (* Status DC bus-a iz state dekodera. *)
	END_VAR
	VAR_OUTPUT (* Izlazi statusa izvrsenja i zadavanja frekvencije. *)
		out_BUSY : {REDUND_UNREPLICABLE} BOOL; (* TRUE kada je komanda u tranziciji. *)
		set_freq : INT; (* Izracunata/odobrena izlazna frekvencija. *)
		out_DONE : {REDUND_UNREPLICABLE} BOOL; (* TRUE kada je komanda zavrsena. *)
	END_VAR
	VAR (* Interne reference i pomocne promenljive upravljanja. *)
		en : {REDUND_UNREPLICABLE} BOOL; (* Legacy enable medjupromenljiva. *)
		ref_ctrlWord : REFERENCE TO UINT; (* Referenca na komandnu rec ATV mapiranja. *)
	END_VAR
END_FUNCTION_BLOCK
```

#### fbCheckStateCanOpenENC.st
```iecst
(* Dekodiranje CANopen ENC status reci u standardni state kod. *)
FUNCTION_BLOCK fbCheckStateCanOpenENC
	(* ---------------------------------------------------------------------- *)
	(* Referentna mapa bitova status reci (ENC):                               *)
	(* b0=bus voltage, b1=run effective, b2=jog effective, b3=running,         *)
	(* b4=aktuelni smer reverse, b5=zadati smer reverse,                        *)
	(* b6=deceleration braking, b7=acceleration, b8=deceleration,              *)
	(* b9=alarm, b10=fault, b11=current limit, b12=fault self recovery,        *)
	(* b13=self tuning, b14=free stop, b15=speed tracking start.               *)
	(* ---------------------------------------------------------------------- *)

	(* ---------------------------------------------------------------------- *)
	(* 1) Povezivanje status reci preko adrese                               *)
	(* ---------------------------------------------------------------------- *)
	ref_statusWord ACCESS in_addr_StatusWord;

	(* ---------------------------------------------------------------------- *)
	(* 2) Prioritetna dekodiranja stanja (alarm/fault/tuning/operacija)      *)
	(* ---------------------------------------------------------------------- *)
	IF (ref_statusWord.9 = 1) THEN
		out_State := ST_ALARM; (* Alarm bit aktivan. *)
	ELSIF (ref_statusWord.10 = 1) OR (ref_statusWord.12 = 1) THEN
		out_State := ST_FAULT; (* Fault ili self-recovery fault signal. *)
	ELSIF (ref_statusWord.13 = 1) THEN
		out_State := ST_TUNING; (* Samopodesavanje aktivno. *)
	ELSIF (ref_statusWord.0 = 0) THEN
		out_State := ST_PWR_OFF; (* Nema bus napona. *)
	ELSIF (ref_statusWord = 1) THEN
		out_State := ST_READY; (* Osnovno ready stanje. *)
	ELSIF (ref_statusWord.14 = 1) OR (ref_statusWord.6 = 1) OR (ref_statusWord.8 = 1) THEN
		out_State := ST_STOPPING; (* Free stop/deceleration uslovi. *)
	ELSIF (ref_statusWord.7 = 1) THEN
		out_State := ST_PREOPERATIONAL; (* Ubrzavanje/tranzicija pre stabilnog rada. *)
	ELSIF (ref_statusWord.2 = 1) THEN
		out_State := ST_JOG; (* Jog komanda efektivna. *)
	ELSIF (ref_statusWord.3 = 1) AND (ref_statusWord.1 = 1) THEN
		out_State := ST_RUN; (* Kontinualni rad potvrden. *)
	END_IF;

END_FUNCTION_BLOCK
```

#### fbControlCanOpenENC.st
```iecst
(* Kontrola CANopen ENC varijante kroz CtrlWord sekvencu. *)
FUNCTION_BLOCK fbControlCanOpenENC

	(* ---------------------------------------------------------------------- *)
	(* 1) Povezivanje mapiranih reci preko adresa                              *)
	(* ---------------------------------------------------------------------- *)
	ref_statusWord ACCESS in_addr_StatusWord;
	ref_ctrlWord ACCESS in_addr_CtrlWord;
	r_ctrlWord ACCESS in_addr_r_CtrlWord;

	(* ---------------------------------------------------------------------- *)
	(* 2) Interna enable priprema                                               *)
	(* ---------------------------------------------------------------------- *)
	IF cmd.Enable THEN
		en := 1;
	ELSE
		en := 0;
	END_IF;

	(* ---------------------------------------------------------------------- *)
	(* 3) Komandna sekvenca u aktivnom bus stanju                              *)
	(* ---------------------------------------------------------------------- *)
	IF en AND (ref_statusWord.0 = 1) THEN

		IF (ref_statusWord.1 = 0) AND (ref_statusWord.2 = 0) THEN

			IF (ref_ctrlWord = 6) AND  ref_statusWord.8 = 0  AND NOT(cmd.Stop) THEN
				ref_ctrlWord := 6;
			END_IF;

			IF cmd.Jog_fwd AND NOT(out_BUSY) THEN
				ref_ctrlWord := 3;
				out_BUSY := TRUE;
				out_DONE := FALSE;
			END_IF;

			IF cmd.Jog_rev AND NOT(out_BUSY) THEN
				ref_ctrlWord := 4;
				out_BUSY := TRUE;
				out_DONE := FALSE;
			END_IF;

			IF cmd.Run_fwd AND NOT(out_BUSY) THEN
				ref_ctrlWord := 7;
				out_BUSY := TRUE;
				out_DONE := FALSE;
			END_IF;

			IF cmd.Run_rev AND NOT(out_BUSY) THEN
				ref_ctrlWord := 8;
				out_BUSY := TRUE;
				out_DONE := FALSE;
			END_IF;

		ELSE

			IF cmd.Jog_fwd AND (ref_statusWord.2 = 1) THEN
				out_BUSY := FALSE;
				out_DONE := TRUE;
			ELSIF cmd.Jog_rev AND (ref_statusWord.2 = 1) THEN
				out_BUSY := FALSE;
				out_DONE := TRUE;
			ELSIF (ref_statusWord.2 = 1) THEN
				ref_ctrlWord := 6;
			END_IF;

			IF cmd.Run_fwd AND (ref_statusWord.1 = 1) THEN
				out_BUSY := FALSE;
				out_DONE := TRUE;
			ELSIF cmd.Run_rev AND (ref_statusWord.1 = 1) THEN
				out_BUSY := FALSE;
				out_DONE := TRUE;
			ELSIF (ref_statusWord.1 = 1) THEN
				ref_ctrlWord := 6;
			END_IF;
			IF NOT(cmd.Jog_fwd) AND NOT(cmd.Jog_rev) AND NOT(cmd.Stop) AND NOT(cmd.Run_fwd) AND NOT(cmd.Run_rev) THEN
				ref_ctrlWord := 6;
			END_IF;

		END_IF;

		(* Stop komanda ima prioritet nad run/jog namerom. *)
		IF cmd.Stop THEN
			ref_ctrlWord := 6;
			(* Legacy alternativa sa toggle 0/6 je uklonjena iz aktivne logike. *)
		END_IF;

		(* Rucni reset fault uslova. *)
		IF cmd.Reset THEN
			ref_ctrlWord := 9;
			out_BUSY := FALSE;
			out_DONE := TRUE;
		END_IF;

		IF NOT(cmd.Reset) AND NOT(cmd.Jog_fwd) AND NOT(cmd.Jog_rev) AND NOT(cmd.Stop) AND NOT(cmd.Run_fwd) AND NOT(cmd.Run_rev) THEN
			out_BUSY := FALSE;
			out_DONE := FALSE;
		END_IF;
	ELSE
		(* ------------------------------------------------------------------ *)
		(* 4) Fallback kada nije enable ili nema bus napona                    *)
		(* ------------------------------------------------------------------ *)
		ref_ctrlWord := 6;

		IF cmd.Reset THEN
			ref_ctrlWord := 9;
		END_IF;

		out_BUSY := FALSE;
		out_DONE := FALSE;
	END_IF;

	(* ---------------------------------------------------------------------- *)
	(* 5) Auto-reset sekvenca nakon detekcije fault/self-recovery signala      *)
	(* ---------------------------------------------------------------------- *)
	IF cmd.en_autoReset THEN
		IF  NOT(ref_ctrlWord = 3) AND  (r_ctrlWord = 3) THEN

			IF start_check THEN
	  			ref_ctrlWord := 9;
				start_check := FALSE;
			ELSE
				ref_ctrlWord := 6;
				start_check := TRUE;
			END_IF;
		END_IF;
	END_IF;

END_FUNCTION_BLOCK
```

#### fbCheckStateCanOpenATV.st
```iecst
(* Dekodiranje ATV status reci u ATV state kod i DC bus status. *)
FUNCTION_BLOCK fbCheckStateCanOpenATV

	(* ---------------------------------------------------------------------- *)
	(* 1) Povezivanje status reci preko adrese                               *)
	(* ---------------------------------------------------------------------- *)
	ref_statusWord ACCESS in_addr_StatusWord;

	(* ---------------------------------------------------------------------- *)
	(* 2) Prioritetna dekodiranja ATV stanja                                  *)
	(* ---------------------------------------------------------------------- *)
	IF (ref_statusWord.3 = TRUE) THEN
		IF(ref_statusWord.0 = FALSE) AND (ref_statusWord.1 = FALSE) AND (ref_statusWord.2 = FALSE) THEN
			out_State := STATV_ERR; (* Hard error stanje. *)
		ELSE
			out_State := STATV_ERR_MNG; (* Error management aktivan. *)
		END_IF;

	ELSIF (ref_statusWord.6 = TRUE) THEN
		out_State := STATV_SWH_DISABLE; (* Switch disable stanje. *)

	ELSIF (ref_statusWord.5 = FALSE) THEN
		IF(ref_statusWord.0 = TRUE) AND (ref_statusWord.1 = TRUE) AND (ref_statusWord.2 = TRUE) THEN
			out_State := STATV_FAST_STOP; (* Fast stop stanje. *)
		ELSE
			out_State := STATV_RDY_NOT; (* Nije ready. *)
		END_IF;

	ELSIF (ref_statusWord.2 = TRUE) THEN
		out_State := STATV_RUN; (* Run stanje. *)

	ELSIF (ref_statusWord.1 = TRUE) THEN
		out_State := STATV_SWH_ON; (* Switched on stanje. *)

	ELSIF (ref_statusWord.0 = FALSE) THEN
		out_State := STATV_RDY_NOT; (* Nije spreman za rad. *)

	ELSIF (ref_statusWord.0 = TRUE) THEN
		out_State := STATV_RDY; (* Ready stanje. *)
		DC_BUS_ON := ref_statusWord.4; (* U ready stanju preuzima se DC bus bit. *)
	END_IF;

END_FUNCTION_BLOCK
```

#### fbControlCanOpenATV.st
```iecst
(* Kontrola ATV CANopen varijante kroz state-zavisnu CtrlWord logiku. *)
FUNCTION_BLOCK fbControlCanOpenATV

	(* ---------------------------------------------------------------------- *)
	(* 1) Povezivanje komandne reci preko adrese                               *)
	(* ---------------------------------------------------------------------- *)
	ref_ctrlWord ACCESS in_addr_CtrlWord;

	(* FastStop se tretira prioritetno kad nije vec u switch-disable stanju. *)
	IF(cmd.FastStop = TRUE) AND NOT(StatusWord = STATV_SWH_DISABLE) THEN
		ref_ctrlWord := 2;
		set_freq := 0;
	END_IF;

	(* ---------------------------------------------------------------------- *)
	(* 2) State-zavisna obrada komandi                                         *)
	(* ---------------------------------------------------------------------- *)
	CASE StatusWord OF

		STATV_PWR_OFF:
			(* Nema aktivne akcije dok je pogon bez napajanja. *)

		STATV_RDY_NOT:
			(* Pogon nije ready; ceka se validan prelaz stanja iz drive-a. *)

		STATV_SWH_DISABLE:

			IF (cmd.Enable = TRUE) THEN
				ref_ctrlWord := 6; (* Prelaz ka ready sekvenci. *)
			END_IF

		STATV_RDY:

			IF(DC_BUS_STATE = TRUE) AND (cmd.Enable) THEN
				ref_ctrlWord := 7; (* Uslovi ispunjeni za switch-on. *)
			END_IF
			IF (cmd.Enable = FALSE) THEN
				ref_ctrlWord := 0;
			END_IF

		STATV_SWH_ON:
			IF(cmd.Run_fwd = TRUE) AND (cmd.Enable = TRUE) THEN
				ref_ctrlWord := 15;
				ref_ctrlWord.11 := FALSE;
				ref_ctrlWord.12 := TRUE;
			ELSIF (cmd.Run_rev = TRUE) AND (cmd.Enable = TRUE) THEN
				ref_ctrlWord := 15;
				ref_ctrlWord.12 := FALSE;
				ref_ctrlWord.11 := TRUE;
			ELSIF (cmd.Enable = FALSE) THEN
				ref_ctrlWord := 0;
			END_IF

		STATV_RUN:

			IF(cmd.FastStop = TRUE) THEN
				ref_ctrlWord := 2;
				set_freq := 0;
			ELSIF(cmd.Enable = FALSE) THEN
				ref_ctrlWord := 0;
				set_freq := 0;
				ref_ctrlWord.8 := cmd.Stop;

			ELSIF ((cmd.Run_fwd = FALSE) AND (cmd.Run_rev = FALSE)) OR cmd.Stop THEN
				ref_ctrlWord := 7;
				set_freq := 0;
			ELSE
				set_freq := in_set_freq;
			END_IF

		STATV_FAST_STOP:

			IF (cmd.FastStop = FALSE) THEN
				ref_ctrlWord := 0;
				set_freq := 0;
				cmd.Run_fwd := FALSE;
				cmd.Run_rev := FALSE;
				cmd.Stop := FALSE;
				(* Legacy napomena: cmd.Enable se namerno ne resetuje automatski. *)
			END_IF;

			(* STATV_ERR_MNG je obradjen kroz state dekoder i mapiranje u glavnom FB-u. *)

		STATV_ERR:

			IF (cmd.Reset = TRUE) THEN
				cmd.Run_fwd := FALSE;
				cmd.Run_rev := FALSE;
				cmd.Stop := FALSE;
				(* Legacy napomena: cmd.Enable se namerno ne resetuje automatski. *)
				ref_ctrlWord := 128;
				set_freq := 0;
			END_IF;
	END_CASE

END_FUNCTION_BLOCK
```
